# B&R Automation Studio project NAEUL004C00R13L518F00 (part 47)

### LF.typ - Do Not Change!!!
```iecst
(*2019-04-25*)
(**)
(*Action*)

TYPE
	eLFAction :
		(
		LFActIdle,
		LFActBGStartRun,
		LFActBGStopRun,
		LFActSyncPLCTm,
		LFActChgAllAuto,
		LFActChgAllMnl,
		LFActChgSeqAuto,
		LFActChgSeqMnl
		);
	eLFOPCUAStep :
		(
		LFOPCUAStepIncCntr,
		LFOPCUAStepChkHdls,
		LFOPCUAStepConnect,
		LFOPCUAStepWriteHdls,
		LFOPCUAStepReadHdls,
		LFOPCUAStepWrite,
		LFOPCUAStepRead,
		LFOPCUAStepStopChk
		);
	tyOPCUAHdlList : 	STRUCT
		a_dwHdls : ARRAY[0..MAX_INDEX_NODELIST]OF DWORD;
	END_STRUCT;
END_TYPE

(* *)

TYPE
	tyLFLeader1 : 	STRUCT
		In : tyLFLeaderIn1;
		Out : tyLFLeaderOut1;
	END_STRUCT;
	tyLFLeaderIn1 : 	STRUCT
		bPrep : BOOL;
		bEn : BOOL;
		bDis : BOOL;
	END_STRUCT;
	tyLFLeaderOut1 : 	STRUCT
		eStat : eLFAction;
		eStatus : eFBStatus;
		sStatTxt : STRING[100];
		a_tyFollowerInfo : ARRAY[1..c_diLFClntNum]OF tyLFFollowerInfo;
		a_tyFollowerToLeaderTag : ARRAY[1..c_diLFClntNum]OF tyLFFollowerToLeaderTag;
		tyAlmData : tyAlmDat;
	END_STRUCT;
END_TYPE

(* *)

TYPE
	tyLFFollower1 : 	STRUCT
		In : tyLFFollowerIn1;
		Out : tyLFFollowerOut1;
	END_STRUCT;
	tyLFFollowerIn1 : 	STRUCT
		bEn : BOOL;
		bDis : BOOL;
		bPrep : BOOL;
		bUSWidthChkSen : BOOL;
		bDSWidthChkSen : BOOL;
		sProgNm : STRING[15];
		sMagRcpNm : STRING[15];
	END_STRUCT;
	tyLFFollowerOut1 : 	STRUCT
		eStatus : eFBStatus;
		tyAlmData : tyAlmDat;
		tyInfoData : tyAlmDat;
		tyInfoData1 : tyAlmDat;
		bUSAllow : BOOL;
		bDSAllow : BOOL;
		bProdAccDataMnl : BOOL;
		bProdUpdtDataMnl : BOOL;
		bMagAccDataMnl : BOOL;
		eTimeAct : eTimeAction;
		dtTm : DATE_AND_TIME;
		bWaitRlsBrd : BOOL;
		tyUpdtProdRcp : tyProdRcpParam;
		bLdrSeqCtrlInActive : BOOL;
		tyLeaderInfo : tyLFLeaderInfo;
	END_STRUCT;
END_TYPE
```

### LF.var - Change By Project
```iecst
VAR
	p_LFLeader : UDINT;
	p_LFFollower : UDINT;
	p_Follower1 : UDINT;
	p_Follower2 : UDINT;
	g_sLFLeaderProgNm : STRING[15];
END_VAR
```

### Program Logical/LF/LFLeader (IEC, version 1.00.0) - 1.00.0 - NtHermes v5.00.0 , NtTCP v5.00.0 , NtMessage v5.00.0

#### Init.st - Change By Project
```iecst
(** 2019-04-30 **)
PROGRAM _INIT
	p_LFLeader := ADR(tylocalLFLeader.Out);

END_PROGRAM
```

#### Act_InputConfig.st - Change By Project
```iecst
ACTION Act_InputConfig:

	tylocalLFLeader.In.bPrep	:= g_tyNtParamCurr.bLFPrep;
	tylocalLFLeader.In.bDis 	:= g_tyStartUp.bRun OR (NOT g_tyNtParamCurr.bLFUsrSetPrep AND NOT g_tyNtParamCurr.bLeaderMc) OR (g_tyNtParamCurr.bLFUsrSetPrep AND NOT g_tyMcParamCurr.bLFLeaderMc);
	tylocalLFLeader.In.bEn		:= g_tyMcParamCurr.bLFLeaderMc;

	p_eAct ACCESS p_UILFLeaderAct;
	p_sReqProdRcpNm ACCESS p_ProdRcpCurrRcp0Nm;

	IF g_tyNtParamCurr.bLFProdWidth2Prep THEN
		p_diReqProdWidth ACCESS p_ProdRcpCurrRcp0Width2;
	ELSE
		p_diReqProdWidth ACCESS p_ProdRcpCurrRcp0Width;
	END_IF

	IF (g_tyUIOut.bUILeaderRun = TRUE) AND ((bRun1 = FALSE) OR (bRun2 = FALSE)) THEN
		bUILeaderStart	:= TRUE;
		bUILeaderStop	:= FALSE;
	END_IF

	IF (g_tyUIOut.bUILeaderRun = FALSE) AND ((bRun1 = TRUE) OR (bRun2 = TRUE)) THEN
		bUILeaderStart	:= FALSE;
		bUILeaderStop	:= TRUE;
	END_IF

	IF bUILeaderStart = TRUE THEN
		p_eAct	:= LFActBGStartRun;

		IF (tylocalLFLeader.Out.eStat = LFActBGStartRun) AND (tylocalLFLeader.Out.eStatus = Done) THEN
			p_eAct			:= LFActIdle;
			bUILeaderStart	:= FALSE;
		END_IF

	ELSIF bUILeaderStop = TRUE THEN
		p_eAct	:= LFActBGStopRun;

		IF (tylocalLFLeader.Out.eStat = LFActBGStopRun) AND (tylocalLFLeader.Out.eStatus = Done) THEN
			p_eAct			:= LFActIdle;
			bUILeaderStop	:= FALSE;
		END_IF

	END_IF
END_ACTION
```

#### Act_InitLocal.st - Do Not Change!!!
```iecst
(** 2020-08-06 **)
ACTION Act_InitLocal:

	//Input Reference Link To Local Variable
	p_eAct ACCESS ADR(eAct);

	p_sReqProdRcpNm ACCESS ADR(sReqProdRcpNm);
	p_diReqProdWidth ACCESS ADR(diReqProdWidth);
	p_sReqMagRcpNm ACCESS ADR(sReqMagRcpNm);

	p_sLeaderProgTagNm ACCESS ADR(sLeaderProgTagNm);
	p_sFollowerProgTagNm ACCESS ADR(sFollowerProgTagNm);

	p_bWidth2Prep ACCESS ADR(bWidth2Prep);
	p_bLFSeqStayActive ACCESS ADR(bLFSeqStayActive);

END_ACTION
```

#### Act_Initial.st - Do Not Change!!!
```iecst
ACTION Act_Initial:

	//Initial
	tylocalLFLeader.Out.sStatTxt	:= a_sStatText[tylocalLFLeader.Out.eStat];

	fbOnlineChk.pa_tyLeaderToFollowerTag	:= ADR(a_tyLeaderToFollowerTag);
	fbOnlineChk.pa_tyFollowerInfo	:= ADR(a_tyFollowerInfo);
	fbOnlineChk.tDlyTm				:= g_tyNtParamCurr.tLFLeaderOnlineChkDlyTm;
	fbOnlineChk(bEn := FALSE);

	fbSyncTm.pa_tyLeaderToFollowerTag	:= ADR(a_tyLeaderToFollowerTag);
	fbSyncTm.tDlyTm						:= g_tyNtParamCurr.tLFLeaderSetTmOffDlyTm;
	fbSyncTm(bEn := FALSE);

	fbChgAll.pa_tyLeaderToFollowerTag	:= ADR(a_tyLeaderToFollowerTag);
	fbChgAll(bEn := FALSE);

	fbChgSeq.pa_tyLeaderToFollowerTag	:= ADR(a_tyLeaderToFollowerTag);
	fbChgSeq(bEn := FALSE);

	fbBlkUSDS.pa_tyLeaderToFollowerTag	:= ADR(a_tyLeaderToFollowerTag);
	fbBlkUSDS(bEn := FALSE);

	fbDataUpdt.pa_tyLeaderToFollowerTag	:= ADR(a_tyLeaderToFollowerTag);
	fbDataUpdt(bEn := FALSE);

	fbConnect.tyOPCUAParam.sPort	:= '4840';
	fbConnect(bEn := FALSE);

	fbGetNodeHdlListWr.uiTagNmCnt			:= 17;
	fbGetNodeHdlListWr.a_sServerTagNm[0]	:= CONCAT(CONCAT('::' , p_sFollowerProgTagNm) , ':tyLeaderToFollowerTag.sReqProdRcpNm');
	fbGetNodeHdlListWr.a_sServerTagNm[1]	:= CONCAT(CONCAT('::' , p_sFollowerProgTagNm) , ':tyLeaderToFollowerTag.diReqProdRcpWidth');
	fbGetNodeHdlListWr.a_sServerTagNm[2]	:= CONCAT(CONCAT('::' , p_sFollowerProgTagNm) , ':tyLeaderToFollowerTag.sReqMagRcpNm');
	fbGetNodeHdlListWr.a_sServerTagNm[3]	:= CONCAT(CONCAT('::' , p_sFollowerProgTagNm) , ':tyLeaderToFollowerTag.bMnlAccData');
	fbGetNodeHdlListWr.a_sServerTagNm[4]	:= CONCAT(CONCAT('::' , p_sFollowerProgTagNm) , ':tyLeaderToFollowerTag.bBypassMnlAccData');
	fbGetNodeHdlListWr.a_sServerTagNm[5]	:= CONCAT(CONCAT('::' , p_sFollowerProgTagNm) , ':tyLeaderToFollowerTag.bBlkDS');
	fbGetNodeHdlListWr.a_sServerTagNm[6]	:= CONCAT(CONCAT('::' , p_sFollowerProgTagNm) , ':tyLeaderToFollowerTag.bBlkUS');
	fbGetNodeHdlListWr.a_sServerTagNm[7]	:= CONCAT(CONCAT('::' , p_sFollowerProgTagNm) , ':tyLeaderToFollowerTag.bSetTm');
	fbGetNodeHdlListWr.a_sServerTagNm[8]	:= CONCAT(CONCAT('::' , p_sFollowerProgTagNm) , ':tyLeaderToFollowerTag.dtTm');
	fbGetNodeHdlListWr.a_sServerTagNm[9]	:= CONCAT(CONCAT('::' , p_sFollowerProgTagNm) , ':tyLeaderToFollowerTag.uiTmZone');
	fbGetNodeHdlListWr.a_sServerTagNm[10]	:= CONCAT(CONCAT('::' , p_sFollowerProgTagNm) , ':tyLeaderToFollowerTag.bBypassWidthChk');
	fbGetNodeHdlListWr.a_sServerTagNm[11]	:= CONCAT(CONCAT('::' , p_sFollowerProgTagNm) , ':tyLeaderToFollowerTag.usiRunTm');
	fbGetNodeHdlListWr.a_sServerTagNm[12]	:= CONCAT(CONCAT('::' , p_sFollowerProgTagNm) , ':tyLeaderToFollowerTag.bProdNameUSWarn');
	fbGetNodeHdlListWr.a_sServerTagNm[13]	:= CONCAT(CONCAT('::' , p_sFollowerProgTagNm) , ':tyLeaderToFollowerTag.bProdNameDSWarn');
	fbGetNodeHdlListWr.a_sServerTagNm[14]	:= CONCAT(CONCAT('::' , p_sFollowerProgTagNm) , ':tyLeaderToFollowerTag.bProdWidthUSWarn');
	fbGetNodeHdlListWr.a_sServerTagNm[15]	:= CONCAT(CONCAT('::' , p_sFollowerProgTagNm) , ':tyLeaderToFollowerTag.bProdWidthDSWarn');
	fbGetNodeHdlListWr.a_sServerTagNm[16]	:= CONCAT(CONCAT('::' , p_sFollowerProgTagNm) , ':tyLeaderToFollowerTag.bLeaderSeqCtrlInActive');
	fbGetNodeHdlListWr(bEn := FALSE);

	fbGetNodeHdlListRd.uiTagNmCnt			:= 14;
	fbGetNodeHdlListRd.a_sServerTagNm[0]	:= CONCAT(CONCAT('::' , p_sFollowerProgTagNm) , ':tyFollowerToLeaderTag.sCurrProdRcp');
	fbGetNodeHdlListRd.a_sServerTagNm[1]	:= CONCAT(CONCAT('::' , p_sFollowerProgTagNm) , ':tyFollowerToLeaderTag.diCurrProdWidthUS');
	fbGetNodeHdlListRd.a_sServerTagNm[2]	:= CONCAT(CONCAT('::' , p_sFollowerProgTagNm) , ':tyFollowerToLeaderTag.sCurrMagRcp');
	fbGetNodeHdlListRd.a_sServerTagNm[3]	:= CONCAT(CONCAT('::' , p_sFollowerProgTagNm) , ':tyFollowerToLeaderTag.sIPAddr');
	fbGetNodeHdlListRd.a_sServerTagNm[4]	:= CONCAT(CONCAT('::' , p_sFollowerProgTagNm) , ':tyFollowerToLeaderTag.sMcNm');
	fbGetNodeHdlListRd.a_sServerTagNm[5]	:= CONCAT(CONCAT('::' , p_sFollowerProgTagNm) , ':tyFollowerToLeaderTag.bSectionLeader');
	fbGetNodeHdlListRd.a_sServerTagNm[6]	:= CONCAT(CONCAT('::' , p_sFollowerProgTagNm) , ':tyFollowerToLeaderTag.usiRunTm');
	fbGetNodeHdlListRd.a_sServerTagNm[7]	:= CONCAT(CONCAT('::' , p_sFollowerProgTagNm) , ':tyFollowerToLeaderTag.bProdRcpErr');
	fbGetNodeHdlListRd.a_sServerTagNm[8]	:= CONCAT(CONCAT('::' , p_sFollowerProgTagNm) , ':tyFollowerToLeaderTag.bProdWidthErr');
	fbGetNodeHdlListRd.a_sServerTagNm[9]	:= CONCAT(CONCAT('::' , p_sFollowerProgTagNm) , ':tyFollowerToLeaderTag.bMagRcpErr');
	fbGetNodeHdlListRd.a_sServerTagNm[10]	:= CONCAT(CONCAT('::' , p_sFollowerProgTagNm) , ':tyFollowerToLeaderTag.bSyncTmErr');
	fbGetNodeHdlListRd.a_sServerTagNm[11]	:= CONCAT(CONCAT('::' , p_sFollowerProgTagNm) , ':tyFollowerToLeaderTag.diCurrProdWidthDS');
	fbGetNodeHdlListRd.a_sServerTagNm[12]	:= CONCAT(CONCAT('::' , p_sFollowerProgTagNm) , ':tyFollowerToLeaderTag.eCurrMachineStat');
	fbGetNodeHdlListRd.a_sServerTagNm[13]	:= CONCAT(CONCAT('::' , p_sFollowerProgTagNm) , ':tyFollowerToLeaderTag.bProdChgOverActive');
	fbGetNodeHdlListRd(bEn := FALSE);

	fbWriteList.uiTagNmCnt	:= 17;
	fbWriteList(bEn := FALSE);

	fbReadList.uiTagNmCnt	:= 14;
	fbReadList(bEn := FALSE);

	fbDisconnect(bEn := FALSE);

END_ACTION
```

#### Act_Main.st - Do Not Change!!!
```iecst
ACTION Act_Main:

		//Set p_eAct
	IF tylocalLFLeader.Out.eStatus = Idle OR tylocalLFLeader.Out.eStatus = Busy OR tylocalLFLeader.Out.eStatus = Done THEN
		tylocalLFLeader.Out.eStat	:= p_eAct;
	END_IF

	IF eStatOld <> tylocalLFLeader.Out.eStat THEN
		fbSyncTm(bEn := FALSE);
		fbChgAll(bEn := FALSE);
		fbChgSeq(bEn := FALSE);

		tylocalLFLeader.Out.sStatTxt	:= a_sStatText[tylocalLFLeader.Out.eStat];

		eStatOld	:= tylocalLFLeader.Out.eStat;

		tylocalLFLeader.Out.eStatus		:= Busy;
	END_IF

	//Main
	CASE tylocalLFLeader.Out.eStat OF

		LFActIdle:
			tylocalLFLeader.Out.eStatus	:= Idle;

		LFActBGStartRun:
			IF tylocalLFLeader.Out.eStatus = Idle OR tylocalLFLeader.Out.eStatus = Busy THEN

				bRun1		:= TRUE;
				bRun2		:= TRUE;
				bStop		:= FALSE;
				bStop1Done	:= FALSE;
				bStop2Done	:= FALSE;
				tylocalLFLeader.Out.eStatus		:= Done;

			END_IF

		LFActBGStopRun:
			IF tylocalLFLeader.Out.eStatus = Idle OR tylocalLFLeader.Out.eStatus = Busy THEN

				tylocalLFLeader.Out.eStatus	:= Busy;

				bStop	:= TRUE;

				IF bStop1Done AND bStop2Done THEN

					bRun1		:= FALSE;
					bRun2		:= FALSE;
					bStop		:= FALSE;
					bStop1Done	:= FALSE;
					bStop2Done	:= FALSE;
					tylocalLFLeader.Out.eStatus		:= Done;

				END_IF

			END_IF

		LFActSyncPLCTm:
			IF tylocalLFLeader.Out.eStatus = Idle OR tylocalLFLeader.Out.eStatus = Busy THEN

				IF bRun1 AND bRun2 THEN
					tylocalLFLeader.Out.eStatus	:= Busy;

					fbSyncTm.dtCurrDT		:= g_tyTime.dtCurrDT;
					fbSyncTm.diMcNum		:= diMcNum;
					fbSyncTm(bEn := TRUE);

					IF fbSyncTm.udiStatus = 0 THEN
						tylocalLFLeader.Out.eStatus	:= Done;
					ELSIF fbSyncTm.udiStatus < 65534 THEN
						tylocalLFLeader.Out.eStatus		:= Error;
						udiStatus	:= fbSyncTm.udiStatus;
					END_IF

				ELSE
					tylocalLFLeader.Out.eStatus		:= Error;
					udiStatus	:= 10000;	//Background Not Running While Calling Sync PLC Tm
				END_IF

			END_IF

		LFActChgAllAuto:
			IF tylocalLFLeader.Out.eStatus = Idle OR tylocalLFLeader.Out.eStatus = Busy THEN

				IF bRun1 AND bRun2 THEN
					tylocalLFLeader.Out.eStatus	:= Busy;

					fbChgAll.bChgAuto					:= TRUE;
					fbChgAll.a_bOnline					:= g_tyMcParamCurr.a_bLFOnline;;
					fbChgAll.a_tyFollowerToLeaderTag	:= a_tyFollowerToLeaderTag;
					fbChgAll.sReqProdRcpNm				:= p_sReqProdRcpNm;
					fbChgAll.diReqProdRcpWidth			:= p_diReqProdWidth;
					fbChgAll.sReqMagRcpNm				:= p_sReqMagRcpNm;
					fbChgAll.diMcNum					:= diMcNum;
					fbChgAll(bEn := TRUE);

					IF fbChgAll.udiStatus = 0 THEN
						tylocalLFLeader.Out.eStatus	:= Done;
					ELSIF fbChgAll.udiStatus < 65534 THEN
						tylocalLFLeader.Out.eStatus		:= Error;
						udiStatus	:= fbChgAll.udiStatus;
					END_IF

				ELSE
					tylocalLFLeader.Out.eStatus		:= Error;
					udiStatus	:= 10001;	//Background Not Running While Changing All Recipe Automatically
				END_IF

			END_IF

		LFActChgAllMnl:
			IF tylocalLFLeader.Out.eStatus = Idle OR tylocalLFLeader.Out.eStatus = Busy THEN

				IF bRun1 AND bRun2 THEN
					tylocalLFLeader.Out.eStatus	:= Busy;

					fbChgAll.bChgAuto					:= FALSE;
					fbChgAll.a_bOnline					:= g_tyMcParamCurr.a_bLFOnline;
					fbChgAll.a_tyFollowerToLeaderTag	:= a_tyFollowerToLeaderTag;
					fbChgAll.sReqProdRcpNm				:= p_sReqProdRcpNm;
					fbChgAll.diReqProdRcpWidth			:= p_diReqProdWidth;
					fbChgAll.sReqMagRcpNm				:= p_sReqMagRcpNm;
					fbChgAll.diMcNum					:= diMcNum;
					fbChgAll(bEn := TRUE);

					IF fbChgAll.udiStatus = 0 THEN
						tylocalLFLeader.Out.eStatus	:= Done;
					ELSIF fbChgAll.udiStatus < 65534 THEN
						tylocalLFLeader.Out.eStatus		:= Error;
						udiStatus	:= fbChgAll.udiStatus;
					END_IF

				ELSE
					tylocalLFLeader.Out.eStatus		:= Error;
					udiStatus	:= 10002;	//Background Not Running While Changing All Recipe Manually
				END_IF

			END_IF

		LFActChgSeqAuto:
			IF tylocalLFLeader.Out.eStatus = Idle OR tylocalLFLeader.Out.eStatus = Busy THEN

				IF bRun1 AND bRun2 THEN
					tylocalLFLeader.Out.eStatus	:= Busy;

					fbChgSeq.bChgAuto					:= TRUE;
					fbChgSeq.a_bOnline					:= g_tyMcParamCurr.a_bLFOnline;;
					fbChgSeq.a_tyFollowerToLeaderTag	:= a_tyFollowerToLeaderTag;
					fbChgSeq.sReqProdRcpNm				:= p_sReqProdRcpNm;
					fbChgSeq.diReqProdRcpWidth			:= p_diReqProdWidth;
					fbChgSeq.sReqMagRcpNm				:= p_sReqMagRcpNm;
					fbChgSeq.diMcNum					:= diMcNum;
					fbChgSeq(bEn := TRUE);

					IF fbChgSeq.udiStatus = 0 THEN
						tylocalLFLeader.Out.eStatus	:= Done;
					ELSIF fbChgSeq.udiStatus < 65534 THEN
						tylocalLFLeader.Out.eStatus		:= Error;
						udiStatus	:= fbChgSeq.udiStatus;
					END_IF

				ELSE
					tylocalLFLeader.Out.eStatus		:= Error;
					udiStatus	:= 10003;	//Background Not Running While Changing Recipe In Sequence Automatically
				END_IF

			END_IF

		LFActChgSeqMnl:
			IF tylocalLFLeader.Out.eStatus = Idle OR tylocalLFLeader.Out.eStatus = Busy THEN

				IF bRun1 AND bRun2 THEN
					tylocalLFLeader.Out.eStatus	:= Busy;

					fbChgSeq.bChgAuto					:= FALSE;
					fbChgSeq.a_bOnline					:= g_tyMcParamCurr.a_bLFOnline;;
					fbChgSeq.a_tyFollowerToLeaderTag	:= a_tyFollowerToLeaderTag;
					fbChgSeq.sReqProdRcpNm				:= p_sReqProdRcpNm;
					fbChgSeq.diReqProdRcpWidth			:= p_diReqProdWidth;
					fbChgSeq.sReqMagRcpNm				:= p_sReqMagRcpNm;
					fbChgSeq.diMcNum					:= diMcNum;
					fbChgSeq(bEn := TRUE);

					IF fbChgSeq.udiStatus = 0 THEN
						tylocalLFLeader.Out.eStatus	:= Done;
					ELSIF fbChgSeq.udiStatus < 65534 THEN
						tylocalLFLeader.Out.eStatus		:= Error;
						udiStatus	:= fbChgSeq.udiStatus;
					END_IF

				ELSE
					tylocalLFLeader.Out.eStatus		:= Error;
					udiStatus	:= 10004;	//Background Not Running While Changing Recipe In Sequence Manually
				END_IF

			END_IF

	END_CASE

END_ACTION
```

#### Act_Background.st - Do Not Change!!!
```iecst
ACTION Act_Background:

	IF EDGEPOS(bRun1 AND bRun2) THEN

		FOR di := 1 TO c_diLFClntNum DO
			IF g_tyMcParamCurr.a_sLFIPAddr[di] = '' THEN
				diMcNum	:= di - 1;
				EXIT;
			END_IF
		END_FOR

	END_IF

	Act_Background_OPCUA;
	Act_Background_Process;
	Act_Background_Disconnect;

END_ACTION
```

#### Act_Background_OPCUA.st - Do Not Change!!!
```iecst
ACTION Act_Background_OPCUA:

	IF bRun1 = TRUE THEN

		CASE eOPCUAStep OF

			LFOPCUAStepIncCntr:
				udiNodeCntr	:= udiNodeCntr + 1;

				IF udiNodeCntr > c_diLFClntNum THEN
					udiNodeCntr	:= 1;
				END_IF

				eOPCUAStep	:= LFOPCUAStepChkHdls;

			LFOPCUAStepChkHdls:
				IF g_tyMcParamCurr.a_sLFIPAddr[udiNodeCntr] <> '' THEN
					IF g_tyMcParamCurr.a_bLFOnline[udiNodeCntr] = TRUE THEN
						IF a_dwConnectionHdl[udiNodeCntr] <> 0 THEN
							IF a_bNodeWr[udiNodeCntr] = TRUE THEN
								IF a_bNodeRd[udiNodeCntr] = TRUE THEN
									eOPCUAStep	:= LFOPCUAStepWrite;
								ELSE
									eOPCUAStep	:= LFOPCUAStepReadHdls;
								END_IF
							ELSE
								eOPCUAStep	:= LFOPCUAStepWriteHdls;
							END_IF
						ELSE
							eOPCUAStep	:= LFOPCUAStepConnect;
						END_IF
					ELSE
						eOPCUAStep	:= LFOPCUAStepIncCntr;
					END_IF
				ELSE
					udiNodeCntr	:= 0;
					eOPCUAStep	:= LFOPCUAStepStopChk;
				END_IF

			LFOPCUAStepConnect:
				fbConnect.tyOPCUAParam.sIPAddr	:= g_tyMcParamCurr.a_sLFIPAddr[udiNodeCntr];
				fbConnect(bEn := TRUE);

				IF fbConnect.udiStatus = 0 THEN
					a_dwConnectionHdl[udiNodeCntr]	:= fbConnect.dwConnectionHdl;
					fbConnect(bEn := FALSE);
					eOPCUAStep	:= LFOPCUAStepWriteHdls;
				ELSIF fbConnect.udiStatus < 65534 THEN
					a_dwConnectionHdl[udiNodeCntr]	:= 0;
					fbConnect(bEn := FALSE);
					eOPCUAStep	:= LFOPCUAStepStopChk;
				END_IF

			LFOPCUAStepWriteHdls:
				fbGetNodeHdlListWr.dwConnectionHdl	:= a_dwConnectionHdl[udiNodeCntr];
				fbGetNodeHdlListWr(bEn := TRUE);

				IF fbGetNodeHdlListWr.udiStatus = 0 THEN
					a_bNodeWr[udiNodeCntr]				:= TRUE;
					a_tyWriteHdls[udiNodeCntr].a_dwHdls	:= fbGetNodeHdlListWr.a_dwNodeHdlList;
					fbGetNodeHdlListWr(bEn := FALSE);
					eOPCUAStep	:= LFOPCUAStepReadHdls;
				ELSIF fbGetNodeHdlListWr.udiStatus < 65534 THEN
					a_bNodeWr[udiNodeCntr]	:= FALSE;
					fbGetNodeHdlListWr(bEn := FALSE);
					eOPCUAStep	:= LFOPCUAStepStopChk;
				END_IF

			LFOPCUAStepReadHdls:
				fbGetNodeHdlListRd.dwConnectionHdl	:= a_dwConnectionHdl[udiNodeCntr];
				fbGetNodeHdlListRd(bEn := TRUE);

				IF fbGetNodeHdlListRd.udiStatus = 0 THEN
					a_bNodeRd[udiNodeCntr]				:= TRUE;
					a_tyReadHdls[udiNodeCntr].a_dwHdls	:= fbGetNodeHdlListRd.a_dwNodeHdlList;
					fbGetNodeHdlListRd(bEn := FALSE);
					eOPCUAStep	:= LFOPCUAStepWrite;
				ELSIF fbGetNodeHdlListRd.udiStatus < 65534 THEN
					a_bNodeRd[udiNodeCntr]	:= FALSE;
					fbGetNodeHdlListRd(bEn := FALSE);
					eOPCUAStep	:= LFOPCUAStepStopChk;
				END_IF

			LFOPCUAStepWrite:
				fbWriteList.dwConnectionHdl		:= a_dwConnectionHdl[udiNodeCntr];
				fbWriteList.a_dwNodeHdlList		:= a_tyWriteHdls[udiNodeCntr].a_dwHdls;
				sNodeCntr						:= UDINT_TO_STRING(udiNodeCntr);
				fbWriteList.a_sClientTagNm[0]	:= CONCAT(CONCAT(CONCAT(CONCAT('::' , p_sLeaderProgTagNm) , ':a_tyLeaderToFollowerTag[') , sNodeCntr) , '].sReqProdRcpNm');
				fbWriteList.a_sClientTagNm[1]	:= CONCAT(CONCAT(CONCAT(CONCAT('::' , p_sLeaderProgTagNm) , ':a_tyLeaderToFollowerTag[') , sNodeCntr) , '].diReqProdRcpWidth');
				fbWriteList.a_sClientTagNm[2]	:= CONCAT(CONCAT(CONCAT(CONCAT('::' , p_sLeaderProgTagNm) , ':a_tyLeaderToFollowerTag[') , sNodeCntr) , '].sReqMagRcpNm');
				fbWriteList.a_sClientTagNm[3]	:= CONCAT(CONCAT(CONCAT(CONCAT('::' , p_sLeaderProgTagNm) , ':a_tyLeaderToFollowerTag[') , sNodeCntr) , '].bMnlAccData');
				fbWriteList.a_sClientTagNm[4]	:= CONCAT(CONCAT(CONCAT(CONCAT('::' , p_sLeaderProgTagNm) , ':a_tyLeaderToFollowerTag[') , sNodeCntr) , '].bBypassMnlAccData');
				fbWriteList.a_sClientTagNm[5]	:= CONCAT(CONCAT(CONCAT(CONCAT('::' , p_sLeaderProgTagNm) , ':a_tyLeaderToFollowerTag[') , sNodeCntr) , '].bBlkDS');
				fbWriteList.a_sClientTagNm[6]	:= CONCAT(CONCAT(CONCAT(CONCAT('::' , p_sLeaderProgTagNm) , ':a_tyLeaderToFollowerTag[') , sNodeCntr) , '].bBlkUS');
				fbWriteList.a_sClientTagNm[7]	:= CONCAT(CONCAT(CONCAT(CONCAT('::' , p_sLeaderProgTagNm) , ':a_tyLeaderToFollowerTag[') , sNodeCntr) , '].bSetTm');
				fbWriteList.a_sClientTagNm[8]	:= CONCAT(CONCAT(CONCAT(CONCAT('::' , p_sLeaderProgTagNm) , ':a_tyLeaderToFollowerTag[') , sNodeCntr) , '].dtTm');
				fbWriteList.a_sClientTagNm[9]	:= CONCAT(CONCAT(CONCAT(CONCAT('::' , p_sLeaderProgTagNm) , ':a_tyLeaderToFollowerTag[') , sNodeCntr) , '].uiTmZone');
				fbWriteList.a_sClientTagNm[10]	:= CONCAT(CONCAT(CONCAT(CONCAT('::' , p_sLeaderProgTagNm) , ':a_tyLeaderToFollowerTag[') , sNodeCntr) , '].bBypassWidthChk');
				fbWriteList.a_sClientTagNm[11]	:= CONCAT(CONCAT(CONCAT(CONCAT('::' , p_sLeaderProgTagNm) , ':a_tyLeaderToFollowerTag[') , sNodeCntr) , '].usiRunTm');
				fbWriteList.a_sClientTagNm[12]	:= CONCAT(CONCAT(CONCAT(CONCAT('::' , p_sLeaderProgTagNm) , ':a_tyLeaderToFollowerTag[') , sNodeCntr) , '].bProdNameUSWarn');
				fbWriteList.a_sClientTagNm[13]	:= CONCAT(CONCAT(CONCAT(CONCAT('::' , p_sLeaderProgTagNm) , ':a_tyLeaderToFollowerTag[') , sNodeCntr) , '].bProdNameDSWarn');
				fbWriteList.a_sClientTagNm[14]	:= CONCAT(CONCAT(CONCAT(CONCAT('::' , p_sLeaderProgTagNm) , ':a_tyLeaderToFollowerTag[') , sNodeCntr) , '].bProdWidthUSWarn');
				fbWriteList.a_sClientTagNm[15]	:= CONCAT(CONCAT(CONCAT(CONCAT('::' , p_sLeaderProgTagNm) , ':a_tyLeaderToFollowerTag[') , sNodeCntr) , '].bProdWidthDSWarn');
				fbWriteList.a_sClientTagNm[16]	:= CONCAT(CONCAT(CONCAT(CONCAT('::' , p_sLeaderProgTagNm) , ':a_tyLeaderToFollowerTag[') , sNodeCntr) , '].bLeaderSeqCtrlInActive');
				fbWriteList(bEn := TRUE);

				IF fbWriteList.udiStatus = 0 THEN
					fbWriteList(bEn := FALSE);
					eOPCUAStep	:= LFOPCUAStepRead;
				ELSIF fbWriteList.udiStatus < 65534 THEN
					fbWriteList(bEn := FALSE);
					eOPCUAStep	:= LFOPCUAStepStopChk;
				END_IF

			LFOPCUAStepRead:
				fbReadList.dwConnectionHdl		:= a_dwConnectionHdl[udiNodeCntr];
				fbReadList.a_dwNodeHdlList		:= a_tyReadHdls[udiNodeCntr].a_dwHdls;
				sNodeCntr						:= UDINT_TO_STRING(udiNodeCntr);
				fbReadList.a_sClientTagNm[0]	:= CONCAT(CONCAT(CONCAT(CONCAT('::' , p_sLeaderProgTagNm) , ':a_tyFollowerToLeaderTag[') , sNodeCntr) , '].sCurrProdRcp');
				fbReadList.a_sClientTagNm[1]	:= CONCAT(CONCAT(CONCAT(CONCAT('::' , p_sLeaderProgTagNm) , ':a_tyFollowerToLeaderTag[') , sNodeCntr) , '].diCurrProdWidthUS');
				fbReadList.a_sClientTagNm[2]	:= CONCAT(CONCAT(CONCAT(CONCAT('::' , p_sLeaderProgTagNm) , ':a_tyFollowerToLeaderTag[') , sNodeCntr) , '].sCurrMagRcp');
				fbReadList.a_sClientTagNm[3]	:= CONCAT(CONCAT(CONCAT(CONCAT('::' , p_sLeaderProgTagNm) , ':a_tyFollowerToLeaderTag[') , sNodeCntr) , '].sIPAddr');
				fbReadList.a_sClientTagNm[4]	:= CONCAT(CONCAT(CONCAT(CONCAT('::' , p_sLeaderProgTagNm) , ':a_tyFollowerToLeaderTag[') , sNodeCntr) , '].sMcNm');
				fbReadList.a_sClientTagNm[5]	:= CONCAT(CONCAT(CONCAT(CONCAT('::' , p_sLeaderProgTagNm) , ':a_tyFollowerToLeaderTag[') , sNodeCntr) , '].bSectionLeader');
				fbReadList.a_sClientTagNm[6]	:= CONCAT(CONCAT(CONCAT(CONCAT('::' , p_sLeaderProgTagNm) , ':a_tyFollowerToLeaderTag[') , sNodeCntr) , '].usiRunTm');
				fbReadList.a_sClientTagNm[7]	:= CONCAT(CONCAT(CONCAT(CONCAT('::' , p_sLeaderProgTagNm) , ':a_tyFollowerToLeaderTag[') , sNodeCntr) , '].bProdRcpErr');
				fbReadList.a_sClientTagNm[8]	:= CONCAT(CONCAT(CONCAT(CONCAT('::' , p_sLeaderProgTagNm) , ':a_tyFollowerToLeaderTag[') , sNodeCntr) , '].bProdWidthErr');
				fbReadList.a_sClientTagNm[9]	:= CONCAT(CONCAT(CONCAT(CONCAT('::' , p_sLeaderProgTagNm) , ':a_tyFollowerToLeaderTag[') , sNodeCntr) , '].bMagRcpErr');
				fbReadList.a_sClientTagNm[10]	:= CONCAT(CONCAT(CONCAT(CONCAT('::' , p_sLeaderProgTagNm) , ':a_tyFollowerToLeaderTag[') , sNodeCntr) , '].bSyncTmErr');
				fbReadList.a_sClientTagNm[11]	:= CONCAT(CONCAT(CONCAT(CONCAT('::' , p_sLeaderProgTagNm) , ':a_tyFollowerToLeaderTag[') , sNodeCntr) , '].diCurrProdWidthDS');
				fbReadList.a_sClientTagNm[12]	:= CONCAT(CONCAT(CONCAT(CONCAT('::' , p_sLeaderProgTagNm) , ':a_tyFollowerToLeaderTag[') , sNodeCntr) , '].eCurrMachineStat');
				fbReadList.a_sClientTagNm[13]	:= CONCAT(CONCAT(CONCAT(CONCAT('::' , p_sLeaderProgTagNm) , ':a_tyFollowerToLeaderTag[') , sNodeCntr) , '].bProdChgOverActive');
				fbReadList(bEn := TRUE);

				IF fbReadList.udiStatus = 0 THEN
					fbReadList(bEn := FALSE);
					eOPCUAStep	:= LFOPCUAStepStopChk;
				ELSIF fbReadList.udiStatus < 65534 THEN
					fbReadList(bEn := FALSE);
					eOPCUAStep	:= LFOPCUAStepStopChk;
				END_IF

			LFOPCUAStepStopChk:
				IF bStop AND bStop2Done THEN
					IF bCntr = FALSE THEN
						bCntr	:= TRUE;
					ELSE
						bStop1Done	:= TRUE;
						bCntr		:= FALSE;
					END_IF
				ELSE
					bCntr	:= FALSE;
				END_IF

				eOPCUAStep	:= LFOPCUAStepIncCntr;

		END_CASE

	END_IF

END_ACTION
```

#### Act_Background_Process.st - Do Not Change!!!
```iecst
ACTION Act_Background_Process:

	IF bRun2 = TRUE AND bStop = FALSE THEN
		fbOnlineChk.a_bOnline				:= g_tyMcParamCurr.a_bLFOnline;
		fbOnlineChk.a_tyFollowerToLeaderTag	:= a_tyFollowerToLeaderTag;
		fbOnlineChk.diMcNum					:= diMcNum;
		fbOnlineChk(bEn := TRUE);

		fbBlkUSDS.a_tyFollowerToLeaderTag	:= a_tyFollowerToLeaderTag;
		fbBlkUSDS.diBeforeOven1			:= g_tyMcParamCurr.diLFMcIdxBeforeOven;
		fbBlkUSDS.diAfterOven1			:= g_tyMcParamCurr.diLFMcIdxAfterOven;
		fbBlkUSDS.diBeforeOven2			:= g_tyMcParamCurr.diLFMcIdxBeforeOven2;
		fbBlkUSDS.diAfterOven2			:= g_tyMcParamCurr.diLFMcIdxAfterOven2;
		fbBlkUSDS.diMcNum				:= diMcNum;
		fbBlkUSDS.pa_bLFOnline			:= g_tyMcParamCurr.a_bLFOnline;
		fbBlkUSDS.bSeqMode				:= (tylocalLFLeader.Out.eStat= LFActChgSeqAuto) OR (tylocalLFLeader.Out.eStat= LFActChgSeqMnl);
		fbBlkUSDS(bEn := TRUE);

		fbDataUpdt.a_bOnline			:= g_tyMcParamCurr.a_bLFOnline;
		fbDataUpdt.diMcNum				:= diMcNum;
		fbDataUpdt(bEn := TRUE);

	ELSIF bStop = TRUE THEN
		fbOnlineChk(bEn := FALSE);
		fbBlkUSDS(bEn := FALSE);
		fbDataUpdt(bEn := FALSE);
		bStop2Done	:= TRUE;

	END_IF

END_ACTION
```

#### Act_Background_Disconnect.st - Do Not Change!!!
```iecst
ACTION Act_Background_Disconnect:

	IF (memcmp(ADR(g_tyMcParamCurr.a_sLFIPAddr) , ADR(a_sLFIPAddrOld) , SIZEOF(a_sLFIPAddrOld)) <> 0) AND (bDisconnecting = FALSE) THEN
		FOR di := 1 TO c_diLFClntNum DO

			IF g_tyMcParamCurr.a_sLFIPAddr[di] <> a_sLFIPAddrOld[di] THEN
				diDisconnectIdx	:= di;
				bDisconnecting	:= TRUE;
				EXIT;
			END_IF

		END_FOR
	END_IF

	IF bDisconnecting = TRUE THEN

		IF a_dwConnectionHdl[diDisconnectIdx] <> 0 THEN
			fbDisconnect.dwConnectionHdl	:= a_dwConnectionHdl[diDisconnectIdx];
			fbDisconnect(bEn := TRUE);

			IF fbDisconnect.udiStatus = 0 THEN
				a_dwConnectionHdl[diDisconnectIdx]	:= 0;
				a_bNodeWr[diDisconnectIdx]			:= FALSE;
				a_bNodeRd[diDisconnectIdx]			:= FALSE;
				memset(ADR(a_tyFollowerToLeaderTag[diDisconnectIdx]) , 0 , SIZEOF(a_tyFollowerToLeaderTag[diDisconnectIdx]));
				fbDisconnect(bEn := FALSE);

				a_sLFIPAddrOld[diDisconnectIdx]	:= g_tyMcParamCurr.a_sLFIPAddr[diDisconnectIdx];
				bDisconnecting						:= FALSE;

			ELSIF fbDisconnect.udiStatus < 65534 THEN
				a_dwConnectionHdl[diDisconnectIdx]	:= 0;
				a_bNodeWr[diDisconnectIdx]			:= FALSE;
				a_bNodeRd[diDisconnectIdx]			:= FALSE;
				memset(ADR(a_tyFollowerToLeaderTag[diDisconnectIdx]) , 0 , SIZEOF(a_tyFollowerToLeaderTag[diDisconnectIdx]));
				fbDisconnect(bEn := FALSE);

				a_sLFIPAddrOld[diDisconnectIdx]	:= g_tyMcParamCurr.a_sLFIPAddr[diDisconnectIdx];
				bDisconnecting						:= FALSE;

			END_IF

		ELSE
			a_bNodeWr[diDisconnectIdx]	:= FALSE;
			a_bNodeRd[diDisconnectIdx]	:= FALSE;
			memset(ADR(a_tyFollowerToLeaderTag[diDisconnectIdx]) , 0 , SIZEOF(a_tyFollowerToLeaderTag[diDisconnectIdx]));

			a_sLFIPAddrOld[diDisconnectIdx]	:= g_tyMcParamCurr.a_sLFIPAddr[diDisconnectIdx];
			bDisconnecting						:= FALSE;

		END_IF

	END_IF

END_ACTION
```

#### Act_Alarm.st - Do Not Change!!!
```iecst
ACTION Act_Alarm:

	IF g_tyRstErrOut.udiRstErr <> udiRstErrOld THEN
		bRstErr			:= TRUE;
		udiRstErrOld	:= g_tyRstErrOut.udiRstErr;
	ELSE
		bRstErr			:= FALSE;
	END_IF

	//Reset Error
	IF (tylocalLFLeader.Out.eStatus = Error) AND bRstErr THEN
		p_eAct	:= LFActIdle;
		tylocalLFLeader.Out.eStat	:= LFActIdle;
	END_IF

	//Error
	IF EDGEPOS(tylocalLFLeader.Out.eStatus = Error) THEN

		tylocalLFLeader.Out.tyAlmData.udiCode		:= udiStatus;
		tylocalLFLeader.Out.tyAlmData.eSeverity		:= AlmSeverityError;
		tylocalLFLeader.Out.tyAlmData.udiRunTime	:= tyAlmData.udiRunTime + 1;
		tylocalLFLeader.Out.tyAlmData.bAlm			:= TRUE;
		tylocalLFLeader.Out.tyAlmData.udiModuleNum  := udiModuleNum;
		g_sLFLeaderProgNm		:= g_tyNtParamCurr.sLFLeaderProgNm;

	ELSIF bRstErr AND (tyAlmData.udiCode <> 0) THEN

		tylocalLFLeader.Out.tyAlmData.udiCode	:= 0;
		tylocalLFLeader.Out.tyAlmData.eSeverity	:= AlmSeverityNA;
		tylocalLFLeader.Out.tyAlmData.bAlm		:= FALSE;
		tylocalLFLeader.Out.sStatTxt	:= a_sStatText[tylocalLFLeader.Out.eStat];

	END_IF

END_ACTION
```

#### Local.var - Do Not Change!!!
```iecst
(*Reference Data Points*)
VAR
	p_eAct : REFERENCE TO eLFAction;
	p_sReqProdRcpNm : REFERENCE TO STRING[254];
	p_diReqProdWidth : REFERENCE TO DINT;
	p_sReqMagRcpNm : REFERENCE TO STRING[15];
	p_sLeaderProgTagNm : REFERENCE TO STRING[15];
	p_sFollowerProgTagNm : REFERENCE TO STRING[15];
END_VAR
(**)
VAR
	tylocalLFLeader : tyLFLeader1;
	a_sStatText : ARRAY[0..50] OF STRING[200] := ['Idling','Background Starting Operations','Background Stopping Operations','Synchronizing PLC Time','Changing All Recipe Automatically','Changing All Recipe Manually','Changing Recipe In Sequence Automatically','Changing Recipe In Sequence Manually',43('')];
END_VAR
(**)
(*Local Alarm*)
VAR
	tyAlmData : tyAlmDat;
END_VAR
(**)
(*Local Output*)
VAR
	a_tyFollowerInfo : ARRAY[1..c_diLFClntNum] OF tyLFFollowerInfo;
	a_tyFollowerToLeaderTag : ARRAY[1..c_diLFClntNum] OF tyLFFollowerToLeaderTag;
END_VAR
(**)
(*Local Input*)
VAR
	eAct : eLFAction;
	udiStatus : UDINT;
	sReqProdRcpNm : STRING[254];
	diReqProdWidth : DINT;
	sReqMagRcpNm : STRING[15];
	sLeaderProgTagNm : STRING[15] := 'LFLeader';
	sFollowerProgTagNm : STRING[15] := 'LFFollower';
	bUILeaderStart : BOOL;
	bUILeaderStop : BOOL;
END_VAR
(**)
VAR
	bRstErr : BOOL;
	udiRstErrOld : UDINT;
	bInitDone : BOOL;
	bInitialDone : BOOL;
	bRun1 : BOOL;
	bRun2 : BOOL;
	bStop : BOOL;
	bStop1Done : BOOL;
	bStop2Done : BOOL;
	bCntr : BOOL;
	di : DINT;
	diDisconnectIdx : DINT := 1;
	diMcNum : DINT;
	a_sLFIPAddrOld : ARRAY[1..c_diLFClntNum] OF STRING[15];
	bDisconnecting : BOOL;
	eStatOld : eLFAction := LFActIdle;
	a_tyLeaderToFollowerTag : ARRAY[1..c_diLFClntNum] OF tyLFLeaderToFollowerTag;
	fbOnlineChk : fbLFLeaderOnlineChk;
	fbSyncTm : fbLFLeaderSyncTm;
	fbChgAll : fbLFLeaderChgAll;
	fbChgSeq : fbLFLeaderChgSeq;
	fbBlkUSDS : fbLFLeaderBlkUSDS;
	fbDataUpdt : fbLFLeaderDataUpdt;
	udiNodeCntr : UDINT;
	sNodeCntr : STRING[80];
	a_dwConnectionHdl : ARRAY[1..c_diLFClntNum] OF DWORD;
	a_bNodeWr : ARRAY[1..c_diLFClntNum] OF BOOL;
	a_bNodeRd : ARRAY[1..c_diLFClntNum] OF BOOL;
	a_tyWriteHdls : ARRAY[1..c_diLFClntNum] OF tyOPCUAHdlList;
	a_tyReadHdls : ARRAY[1..c_diLFClntNum] OF tyOPCUAHdlList;
	eOPCUAStep : eLFOPCUAStep;
	fbConnect : fbOPCUAConnect;
	fbGetNodeHdlListWr : fbOPCUAGetNodeHdlList;
	fbGetNodeHdlListRd : fbOPCUAGetNodeHdlList;
	fbWriteList : fbOPCUAWriteList;
	fbDisconnect : fbOPCUADisconnect;
	fbReadList : fbOPCUAReadList;
	udiModuleNum : UDINT := 3801;
END_VAR
```

### Program Logical/LF/LFFollower (IEC, version 1.00.0) - 1.00.0 - NtHermes v5.00.0 , NtTCP v5.00.0 , NtMessage v5.00.0

#### Init.st - Change By Project
```iecst
(** 2020-08-06 **)
PROGRAM _INIT

	(* Always Change If Project Change *)

	//Physical Configuration
	bAutoUpdtData	:= TRUE;
	bInternalUse	:= FALSE;

	//Pass Address To Global Address For External Use
	//Action, State & Status
	p_LFFollowerStatus	:= ADR(eStatus);

	//Alarm
	p_LFFollowerAlmData		:= ADR(tyAlmData);
	p_LFFollowerInfoData	:= ADR(tyInfoData);
	p_LFFollowerInfoData1	:= ADR(tyInfoData1);

	//Output
	p_LFFollowerUSAllow			:= ADR(bUSAllow);
	p_LFFollowerDSAllow			:= ADR(bDSAllow);
	p_LFFollowerProdAccDataMnl	:= ADR(bProdAccDataMnl);
	p_LFFollowerProdUpdtDataMnl	:= ADR(bProdUpdtDataMnl);
	p_LFFollowerMagAccDataMnl	:= ADR(bMagAccDataMnl);
	p_LFFollowerTimeAct			:= ADR(eTimeAct);
	p_LFFollowerSetDT			:= ADR(tyLeaderToFollowerTag.dtTm);
	p_LFFollowerWaitRlsBrd		:= ADR(bWaitRlsBrd);
	p_LFFollowerUpdtProdRcp		:= ADR(tyUpdtProdRcp);
	p_LFFollowerLdrSeqCtrlInActive	:= ADR(bLeaderSeqCtrlInActive);

	(* Always Change If Project Change *)

END_PROGRAM
```

#### Act_InputConfig.st - Change By Project
```iecst
(** 2020-09-21 **)
ACTION Act_InputConfig:

	//Pass Data To Internal Use
	p_bUIProdAccData ACCESS p_UIProdAccData;
	p_bUIProdUpdtData ACCESS p_UIProdAccData;
	pa_tyProdRcpList ACCESS p_ProdRcpCurrList;
	p_tyCurrProdRcp ACCESS p_ProdRcpCurrRcp0;
	p_tyDispProdRcp ACCESS p_ProdRcpCurrRcp1;
	p_tyFollower ACCESS p_Follower2;

	//Link bPrep, bEn & bDis
	IF g_tyNtParamCurr.bProjLaneBPrep = FALSE THEN
		tylocalLFFollower.In.bDis	:= g_tyStartUp.bRun OR g_tyMcParamCurr.eUSCommA = McSetCommModHermes;
	ELSE
		tylocalLFFollower.In.bDis	:= g_tyStartUp.bRun OR g_tyMcParamCurr.eUSCommA = McSetCommModHermes OR g_tyMcParamCurr.eUSCommB = McSetCommModHermes;
	END_IF

	//Accept Condition with the relevant Information
	bFollowerInfo	:= tyFollowerToLeaderTag.bProdWidthErr OR bProdRcpErrNotExist OR bProdRcpErrWidthMismatch;

	bLeaderInfo		:= (tyLeaderToFollowerTag.bProdWidthUSWarn OR tyLeaderToFollowerTag.bProdWidthDSWarn
	OR ((tyLeaderToFollowerTag.bProdNameUSWarn OR tyLeaderToFollowerTag.bProdNameDSWarn)
	AND (g_tyNtParamCurr.bAWPrep = TRUE) AND (g_tyMcParamCurr.bAWDis = FALSE) AND (g_tyAW.eStat <>AWActGoWidthOff)));

	//Info Message
	IF bFollowerInfo THEN
		IF tyFollowerToLeaderTag.bProdWidthErr = TRUE OR bProdRcpErrWidthMismatch THEN

			p_sInfoMsg		:= 'Product Recipe Width Does Not Match';
			p_sInfoMsg		:= CONCAT(p_sInfoMsg , '$r$n');
			p_sInfoMsg		:= CONCAT(p_sInfoMsg , 'Check Product Width And');
			p_sInfoMsg		:= CONCAT(p_sInfoMsg , '$r$n');
			p_sInfoMsg		:= CONCAT(p_sInfoMsg , 'Leader Request Width');

		ELSIF bProdRcpErrNotExist THEN

			p_sInfoMsg		:= 'New Product Not Found';
			p_sInfoMsg		:= CONCAT(p_sInfoMsg , '$r$n');
			p_sInfoMsg		:= CONCAT(p_sInfoMsg , 'In Product Recipe List');
			p_sInfoMsg		:= CONCAT(p_sInfoMsg , '$r$n');
			p_sInfoMsg		:= CONCAT(p_sInfoMsg , 'Create New Product');
			p_sInfoMsg		:= CONCAT(p_sInfoMsg , '$r$n');
			p_sInfoMsg		:= CONCAT(p_sInfoMsg , 'In Product Setting');
		END_IF
	ELSE

		IF (tyLeaderToFollowerTag.sReqProdRcpNm<>p_tyCurrProdRcp.sRcpNm) AND (tyLeaderToFollowerTag.sReqProdRcpNm<>'')
			AND bLeaderInfo=FALSE THEN

			p_sInfoMsg		:= 'Leader Request New Recipe';
			p_sInfoMsg		:= CONCAT(p_sInfoMsg , '$r$n');
			p_sInfoMsg		:= CONCAT(p_sInfoMsg , 'Old Recipe Name : ');
			p_sInfoMsg		:= CONCAT(p_sInfoMsg , p_tyDispProdRcp.sRcpNm);
			p_sInfoMsg		:= CONCAT(p_sInfoMsg , '$r$n');
			p_sInfoMsg		:= CONCAT(p_sInfoMsg , 'Old Recipe Width : ');
			sWidthInUMTemp	:= DINT_TO_STRING(p_tyDispProdRcp.diWidthInUM / 1000);
			p_sInfoMsg		:= CONCAT(p_sInfoMsg , sWidthInUMTemp);
			p_sInfoMsg		:= CONCAT(p_sInfoMsg , '$r$n');
			p_sInfoMsg		:= CONCAT(p_sInfoMsg , 'New Recipe Name : ');
			p_sInfoMsg		:= CONCAT(p_sInfoMsg , tyLeaderToFollowerTag.sReqProdRcpNm);
			p_sInfoMsg		:= CONCAT(p_sInfoMsg , '$r$n');
			p_sInfoMsg		:= CONCAT(p_sInfoMsg , 'New Recipe Width : ');
			sWidthInUMTemp	:= DINT_TO_STRING(tyLeaderToFollowerTag.diReqProdRcpWidth / 1000);
			p_sInfoMsg		:= CONCAT(p_sInfoMsg , sWidthInUMTemp);

		ELSIF tyLeaderToFollowerTag.bProdNameUSWarn THEN
			p_sInfoMsg		:= 'US Machine Request New Recipe';
			p_sInfoMsg		:= CONCAT(p_sInfoMsg , '$r$n');
			p_sInfoMsg		:= CONCAT(p_sInfoMsg , 'Old Recipe Name : ');
			p_sInfoMsg		:= CONCAT(p_sInfoMsg , p_tyDispProdRcp.sRcpNm);
			p_sInfoMsg		:= CONCAT(p_sInfoMsg , '$r$n');
			p_sInfoMsg		:= CONCAT(p_sInfoMsg , 'Old Recipe Width : ');
			sWidthInUMTemp	:= DINT_TO_STRING(p_tyDispProdRcp.diWidthInUM / 1000);
			p_sInfoMsg		:= CONCAT(p_sInfoMsg , sWidthInUMTemp);
			p_sInfoMsg		:= CONCAT(p_sInfoMsg , '$r$n');
			p_sInfoMsg		:= CONCAT(p_sInfoMsg , 'New Recipe Name : ');
			p_sInfoMsg		:= CONCAT(p_sInfoMsg , tyLeaderToFollowerTag.sReqProdRcpNm);
			p_sInfoMsg		:= CONCAT(p_sInfoMsg , '$r$n');
			p_sInfoMsg		:= CONCAT(p_sInfoMsg , 'New Recipe Width : ');
			sWidthInUMTemp	:= DINT_TO_STRING(tyLeaderToFollowerTag.diReqProdRcpWidth / 1000);
			p_sInfoMsg		:= CONCAT(p_sInfoMsg , sWidthInUMTemp);

		ELSIF tyLeaderToFollowerTag.bProdNameDSWarn THEN
			p_sInfoMsg		:= 'Different Recipe';
			p_sInfoMsg		:= CONCAT(p_sInfoMsg , '$r$n');
			p_sInfoMsg		:= CONCAT(p_sInfoMsg , 'From DS Machine');
			p_sInfoMsg		:= CONCAT(p_sInfoMsg , '$r$n');
			p_sInfoMsg		:= CONCAT(p_sInfoMsg , 'Current Recipe Name : ');
			p_sInfoMsg		:= CONCAT(p_sInfoMsg , p_tyCurrProdRcp.sRcpNm);
			p_sInfoMsg		:= CONCAT(p_sInfoMsg , '$r$n');
			p_sInfoMsg		:= CONCAT(p_sInfoMsg , 'Current Recipe Width : ');
			sWidthInUMTemp	:= DINT_TO_STRING(p_tyCurrProdRcp.diWidthInUM2 / 1000);
			p_sInfoMsg		:= CONCAT(p_sInfoMsg , sWidthInUMTemp);

		ELSIF tyLeaderToFollowerTag.bProdWidthUSWarn THEN
			p_sInfoMsg		:= 'Product Recipe Width Does Not Match';
			p_sInfoMsg		:= CONCAT(p_sInfoMsg , '$r$n');
			p_sInfoMsg		:= CONCAT(p_sInfoMsg , 'Check Product Width And');
			p_sInfoMsg		:= CONCAT(p_sInfoMsg , '$r$n');
			p_sInfoMsg		:= CONCAT(p_sInfoMsg , 'Leader Request Width');

		ELSIF tyLeaderToFollowerTag.bProdWidthDSWarn THEN
			p_sInfoMsg		:= 'Same Recipe : ';
			p_sInfoMsg		:= CONCAT(p_sInfoMsg , p_tyDispProdRcp.sRcpNm);
			p_sInfoMsg		:= CONCAT(p_sInfoMsg , '$r$n');
			p_sInfoMsg		:= CONCAT(p_sInfoMsg , 'But Different Width');
			p_sInfoMsg		:= CONCAT(p_sInfoMsg , '$r$n');
			p_sInfoMsg		:= CONCAT(p_sInfoMsg , 'With DS Machine');
			p_sInfoMsg		:= CONCAT(p_sInfoMsg , '$r$n');
			p_sInfoMsg		:= CONCAT(p_sInfoMsg , 'Machine Outgoing Width : ');
			sWidthInUMTemp	:= DINT_TO_STRING(p_tyDispProdRcp.diWidthInUM2 / 1000);
			p_sInfoMsg		:= CONCAT(p_sInfoMsg , sWidthInUMTemp);

		END_IF
	END_IF

	//Accept New Recipe Condition (Before Loaded New Recipe)
	IF p_eLinkNtParamProjMag = ULMagDual OR p_eLinkNtParamProjMag = ULMagTriple  THEN
		p_bAccNewRcpCond	:= g_tyOps.bRun;  AND (g_tyPshrConv.bHvBrd = FALSE);
	END_IF

	//Update New Recipe Condition (After Loaded New Recipe)
	p_bUpdtNewRcpCond	:= TRUE;

	IF g_tyAlm.bErr THEN
		eCurrMachineStat := InError;
	ELSE
		IF g_tyAlm.bWarning THEN
			eCurrMachineStat := Warning;
		ELSE
			IF g_tyOps.bRun THEN
				eCurrMachineStat := Run;
			ELSE
				IF g_tyUIOut.bUIManualMod THEN
					eCurrMachineStat := Manual;
				ELSE
					eCurrMachineStat := Stop;
				END_IF
			END_IF
		END_IF
	END_IF

END_ACTION
```

#### Cyclic.st - Do Not Change!!!
```iecst
PROGRAM _CYCLIC

	IF bInitDone = FALSE THEN
		bInitDone	:= TRUE;
		Act_InitLocal;

	ELSIF bInitialDone = FALSE THEN
		IF g_tyStartUp.bNtSettingsLoadDone THEN
			bInitialDone	:= TRUE;
			Act_Initial;
		END_IF

	ELSE

		Act_InputConfig;

		IF (tylocalLFFollower.In.bPrep = TRUE) AND (tylocalLFFollower.In.bEn = TRUE) AND (tylocalLFFollower.In.bDis = FALSE) THEN
			Act_Background;

		ELSE
			Act_Main_Disable;
		END_IF

		Act_Alarm;

	END_IF

END_PROGRAM
```

#### Act_InitLocal.st - Do Not Change!!!
```iecst
ACTION Act_InitLocal:

	p_bUIProdAccData ACCESS ADR(bUIProdAccData);
	p_bUIProdUpdtData ACCESS ADR(bUIProdUpdtData);
	p_bUIMagAccData ACCESS ADR(bUIMagAccData);
	pa_tyProdRcpList ACCESS ADR(a_tyProdRcpList);
	p_tyCurrProdRcp ACCESS ADR(tyCurrProdRcp);
	p_tyDispProdRcp ACCESS ADR(tyDispProdRcp);
	p_sCurrMagRcpNm ACCESS ADR(sCurrMagRcpNm);
	p_bAccNewRcpCond ACCESS ADR(bAccNewRcpCond);
	p_bUpdtNewRcpCond ACCESS ADR(bUpdtNewRcpCond);
	p_bAutoUpdtData ACCESS ADR(bAutoUpdtData);
	p_sInfoMsg ACCESS ADR(sInfoMsg);
	p_bInternalUse ACCESS ADR(bInternalUse);
	p_tyInternalReqProdRcp ACCESS ADR(tyInternalReqProdRcp);
	p_bNewBrdEnteredCond ACCESS ADR(bNewBrdEnteredCond);
	p_bOldBrdExitedCond ACCESS ADR(bOldBrdExitedCond);
	p_bRlsBrd ACCESS ADR(bRlsBrd);
	p_bInternalReqProdRcpDiff ACCESS ADR(bInternalReqProdRcpDiff);
	p_bUpdtProdRcpDiff ACCESS ADR(bUpdtProdRcpDiff);
	p_bRlsBrdProdRcpDiff ACCESS ADR(bRlsBrdProdRcpDiff);

END_ACTION
```

#### Act_Initial.st - Do Not Change!!!
```iecst
ACTION Act_Initial:

	//Initial
	fbFollower.diWidthLimit	:= g_tyNtParamCurr.diLFWidthLimit;
	fbFollower(bEn := FALSE);

	fbOnlineChk.p_tyLeaderInfo		:= ADR(tyLeaderInfo);
	fbOnlineChk.tDlyTm				:= g_tyNtParamCurr.tLFFollowerOnlineChkDlyTm;
	fbOnlineChk(bEn := FALSE);

END_ACTION
```

#### Act_Background.st - Do Not Change!!!
```iecst
ACTION Act_Background:

	IF p_bInternalUse = TRUE THEN
		tyLeaderToFollowerTag.sReqProdRcpNm		:= p_tyInternalReqProdRcp.sRcpNm;

		IF g_tyNtParamCurr.bLFProdWidth2Prep THEN
			tyLeaderToFollowerTag.diReqProdRcpWidth	:= p_tyInternalReqProdRcp.diWidthInUM2;
		ELSE
			tyLeaderToFollowerTag.diReqProdRcpWidth	:= p_tyInternalReqProdRcp.diWidthInUM;
		END_IF
		tyLeaderToFollowerTag.sReqMagRcpNm		:= '';
		tyLeaderToFollowerTag.bMnlAccData		:= FALSE;
		tyLeaderToFollowerTag.bBypassMnlAccData	:= FALSE;
		tyLeaderToFollowerTag.bBlkDS			:= FALSE;
		tyLeaderToFollowerTag.bBlkUS			:= FALSE;
		tyLeaderToFollowerTag.bBypassWidthChk	:= TRUE;
		tyLeaderToFollowerTag.bSetTm			:= FALSE;
		tyLeaderToFollowerTag.dtTm				:= 0;
		tyLeaderToFollowerTag.uiTmZone			:= 0;
		tyLeaderToFollowerTag.usiRunTm			:= 0;
		tyLeaderToFollowerTag.bProdNameUSWarn	:= FALSE;
		tyLeaderToFollowerTag.bProdNameDSWarn	:= FALSE;
		tyLeaderToFollowerTag.bProdWidthUSWarn	:= FALSE;
		tyLeaderToFollowerTag.bProdWidthDSWarn	:= FALSE;
		tyLeaderToFollowerTag.bLeaderSeqCtrlInActive	:= FALSE;
	END_IF

	Act_Background_UpdtData;

	//FB
	fbFollower.tyLeaderToFollowerTag	:= tyLeaderToFollowerTag;
	fbFollower.sMcNm					:= g_tyMcParamCurr.sMcNm;
	fbFollower.sIPAddr					:= g_tyMcParamCurr.sIPAddr;
	fbFollower.bSectionLeader			:= g_tyMcParamCurr.bSectionLeader;
	fbFollower.sCurrProdRcpNm			:= p_tyCurrProdRcp.sRcpNm;
	fbFollower.diCurrProdWidthUS		:= p_tyCurrProdRcp.diWidthInUM;
	fbFollower.diCurrProdWidthDS		:= p_tyCurrProdRcp.diWidthInUM2;
	fbFollower.sCurrMagRcpNm			:= p_sCurrMagRcpNm;
	fbFollower.sUpdtLeaderProdRcpNm		:= p_tyFollower.tyUpdtProdRcp.sRcpNm;
	fbFollower.diUpdtLeaderProdWidthUS	:= p_tyFollower.tyUpdtProdRcp.diWidthInUM;
	fbFollower.diUpdtLeaderProdWidthDS	:= p_tyFollower.tyUpdtProdRcp.diWidthInUM2;
	fbFollower.sUpdtLeaderMagRcpNm		:= tylocalLFFollower.In.sMagRcpNm;
	fbFollower.bMnlAccDat				:= g_tyMcParamCurr.bMnlAccDat;
	fbFollower.bAWEn					:= (g_tyNtParamCurr.bAWPrep = TRUE) AND (g_tyMcParamCurr.bAWDis = FALSE);
	fbFollower.bUSWidthChkEn			:= g_tyNtParamCurr.bUSWidthChkPrep AND g_tyMcParamCurr.bUSWidthChkEn;
	fbFollower.bUSWidthChkSen			:= tylocalLFFollower.In.bUSWidthChkSen;
	fbFollower.bDSWidthChkEn			:= g_tyNtParamCurr.bDSWidthChkPrep AND g_tyMcParamCurr.bDSWidthChkEn;
	fbFollower.bDSWidthChkSen			:= tylocalLFFollower.In.bDSWidthChkSen;
	fbFollower.bProdWidthChk			:= g_tyNtParamCurr.bLFProdWidthChk;
	fbFollower.bProdRcpErr				:= bProdRcpErr;
	fbFollower.bMagRcpErr				:= bMagRcpErr;
	fbFollower.bSetTmErr				:= bSetTmErr;
	fbFollower.eCurrMachineStat			:= eCurrMachineStat;
	fbFollower.bProdChgOverActive		:= (g_tyAW.eStat = AWActGoWidthOff);
	fbFollower.bDBAOnWOAlign			:= g_tyMcParamCurr.bDBAOnWOAlign;

	fbFollower(bEn := TRUE);

	tyFollowerToLeaderTag	:= fbFollower.tyFollowerToLeaderTag;
	bProdAccDataReq			:= fbFollower.bProdAccDataReq OR (p_bInternalReqProdRcpDiff = TRUE) ;
	bMagAccDataReq			:= fbFollower.bMagAccDataReq;
	bAutoAccData			:= fbFollower.bAutoAccData;

	IF p_bInternalUse THEN
		bLeaderOnline			:= TRUE;
	ELSE
		bLeaderOnline			:= tyLeaderInfo.bOnline;
	END_IF

	IF bLeaderOnline=FALSE THEN
		bUSAllow				:= TRUE;
		bDSAllow				:= TRUE;
		bLeaderSeqCtrlInActive	:= FALSE;
	ELSE
		bUSAllow				:= fbFollower.bUSAllow AND (p_bInternalReqProdRcpDiff = FALSE);
		bDSAllow				:= fbFollower.bDSAllow;
		bLeaderSeqCtrlInActive	:= tyLeaderToFollowerTag.bLeaderSeqCtrlInActive;
	END_IF

	fbOnlineChk.tyLeaderToFollowerTag	:= tyLeaderToFollowerTag;
	fbOnlineChk(bEn := TRUE);

	Act_Background_AccData;
	Act_Background_ChkRlsBrd;

	//Set Time
	IF EDGEPOS(tyLeaderToFollowerTag.bSetTm) THEN
		bSetTm	:= TRUE;
	END_IF

	IF bSetTm = TRUE THEN
		eTimeAct	:= TimeActSetTime;

		IF (g_tyTime.eStat = TimeActSetTime) AND (g_tyTime.eMainStatus = Done) THEN
			eTimeAct		:= TimeActIdle;
			bSetTm			:= FALSE;
		ELSIF g_tyTime.eMainStatus = Error THEN
			eTimeAct		:= TimeActIdle;
			bSetTm			:= FALSE;
		END_IF
	END_IF

	bSetTmErr	:= g_tyTime.eMainStatus = Error;

	IF (eStatus = Error) AND bRstErr THEN
		eStatus		:= Idle;
		udiStatus	:= 0;
		bProdRcpErr	:= FALSE;
		bProdRcpErrNotExist	:= FALSE;
		bProdRcpErrWidthMismatch:= FALSE;
		bMagRcpErr	:= FALSE;
	END_IF

END_ACTION
```

#### Act_Background_ChkRlsBrd.st - Do Not Change!!!
```iecst
ACTION Act_Background_ChkRlsBrd:

	IF tyRlsBrdProdRcpNm.sRcpNm = '' THEN
		tyRlsBrdProdRcpNm	:= p_tyCurrProdRcp;

	ELSIF (tyRlsBrdProdRcpNm.sRcpNm <> p_tyCurrProdRcp.sRcpNm) OR (p_bRlsBrdProdRcpDiff = TRUE) THEN

		IF p_bNewBrdEnteredCond = TRUE THEN
			bNewBrdEntered	:= TRUE;
		END_IF

		IF p_bOldBrdExitedCond = TRUE THEN
			bOldBrdExited	:= TRUE;
		END_IF

		IF bNewBrdEntered AND bOldBrdExited THEN
			bWaitRlsBrd	:= TRUE;
		END_IF

		IF bWaitRlsBrd AND p_bRlsBrd THEN
			tyRlsBrdProdRcpNm	:= p_tyCurrProdRcp;
		END_IF

	ELSE
		bNewBrdEntered	:= FALSE;
		bOldBrdExited	:= FALSE;
		bWaitRlsBrd		:= FALSE;

	END_IF

END_ACTION
```

#### Act_Background_UpdtData.st - Do Not Change!!!
```iecst
ACTION Act_Background_UpdtData:

	//Update To Leader Recipe
	CASE usiProdUpdtDatStep OF
		0:
			//Update New Recipe Condition
			IF tyUpdtProdRcp.sRcpNm <> '' THEN
				IF (p_tyCurrProdRcp.sRcpNm <> tyUpdtProdRcp.sRcpNm) OR (p_bUpdtProdRcpDiff = TRUE) THEN
					IF p_bUpdtNewRcpCond = TRUE THEN
						usiProdUpdtDatStep	:= 1;
					END_IF
				END_IF
			ELSE
				tyUpdtProdRcp	:= p_tyCurrProdRcp;
			END_IF

		1:
			//Manual Update Data Check
			IF p_bAutoUpdtData = FALSE THEN
				bProdUpdtDataMnl	:= TRUE;

				IF p_bUIProdUpdtData = TRUE THEN
					bProdUpdtDataMnl	:= FALSE;
					usiProdUpdtDatStep	:= 2;
				END_IF
			ELSE
				bProdUpdtDataMnl	:= FALSE;
				usiProdUpdtDatStep	:= 2;
			END_IF

		2:
			//Update New Recipe
			tyUpdtProdRcp	:= p_tyCurrProdRcp;

			usiProdUpdtDatStep	:= 0;

	END_CASE

END_ACTION
```

#### Act_Background_AccData.st - Do Not Change!!!
```iecst
ACTION Act_Background_AccData:
	//Product Accept Data Request
	CASE usiProdAccDatStep OF
		0:
			//Check Error & Request Accept Data
			// If Product Name/Width Error, Check In Background To Update Data
			IF ((eStatus <> Error) AND (bProdAccDataReq = TRUE)) OR bProdRcpErr THEN
				sReqProdRcpNm		:= tyLeaderToFollowerTag.sReqProdRcpNm;
				diReqProdRcpWidth	:= tyLeaderToFollowerTag.diReqProdRcpWidth;
				usiProdAccDatStep	:= 1;
			END_IF

			IF bLeaderOnline=FALSE THEN
				tyInfoData.udiCode		:= 0;
				tyInfoData.eSeverity	:= AlmSeverityNA;

				bProdRcpErr 			:= FALSE;
				bProdRcpErrNotExist		:= FALSE;
				bProdRcpErrWidthMismatch:= FALSE;
			END_IF

		1:
			IF p_bInternalUse THEN
				usiProdAccDatStep	:= 2;
			ELSE
				//Check In List Of Recipe
				FOR i := 1 TO 2000 DO
					IF sReqProdRcpNm = '' THEN
						EXIT;
					ELSIF sReqProdRcpNm = pa_tyProdRcpList[i].sRcpNm  THEN
						EXIT;
					END_IF
				END_FOR

				IF sReqProdRcpNm = pa_tyProdRcpList[i].sRcpNm AND diReqProdRcpWidth <> pa_tyProdRcpList[i].diWidthInUM THEN
					//Width Mismatch
					bProdRcpErr := TRUE;
					bProdRcpErrWidthMismatch:= TRUE;
					bProdRcpErrNotExist		:= FALSE;
					usiProdAccDatStep	:= 0;
				ELSIF i > 2000 THEN
					//Recipe Not Exist
					bProdRcpErr := TRUE;
					bProdRcpErrNotExist	:= TRUE;
					bProdRcpErrWidthMismatch:= FALSE;
					usiProdAccDatStep	:= 0;
				ELSE
					bProdRcpErr := FALSE;
					bProdRcpErrNotExist	:= FALSE;
					bProdRcpErrWidthMismatch:= FALSE;
					usiProdAccDatStep	:= 2;
				END_IF

				//Info Message
				IF bLeaderOnline=FALSE THEN

					tyInfoData.udiCode		:= 0;
					tyInfoData.eSeverity	:= AlmSeverityNA;

					bProdRcpErr 			:= FALSE;
					bProdRcpErrNotExist		:= FALSE;
					bProdRcpErrWidthMismatch:= FALSE;
				ELSE
					IF p_bInternalUse = FALSE THEN
						IF bLeaderInfo OR bFollowerInfo THEN
//							tyInfoData.sProgNm		:= g_tyNtParamCurr.sLFFollowerProgNm;
							tyInfoData.udiCode		:= 10000;
							tyInfoData.eSeverity	:= AlmSeverityInfo;
							tyInfoData.sAlmMsg		:= p_sInfoMsg;
						ELSE
//							tyInfoData.sProgNm		:= '';
							tyInfoData.udiCode		:= 0;
							tyInfoData.eSeverity	:= AlmSeverityNA;

						END_IF
					ELSE
						IF p_sInfoMsg <> '' THEN
//							tyInfoData.sProgNm		:= g_tyNtParamCurr.sLFFollowerProgNm;
							tyInfoData.udiCode		:= 10000;
							tyInfoData.eSeverity	:= AlmSeverityInfo;
//							tyInfoData.sAlmMsg		:= p_sInfoMsg;
						ELSE
//							tyInfoData.sProgNm		:= '';
							tyInfoData.udiCode		:= 0;
							tyInfoData.eSeverity	:= AlmSeverityNA;
//							tyInfoData.sAlmMsg		:= '';
						END_IF
					END_IF
				END_IF
			END_IF

		2:
			//Manual Accept Data Check
			IF bProdAccDataReq = TRUE THEN
				IF bAutoAccData = FALSE THEN
					bProdAccDataMnl	:= TRUE;

					//Info Message
					IF bLeaderOnline=FALSE THEN
//						tyInfoData.sProgNm		:= '';
						tyInfoData.udiCode		:= 0;
						tyInfoData.eSeverity	:= AlmSeverityNA;
//						tyInfoData.sAlmMsg		:= '';
					ELSE
						IF p_sInfoMsg <> '' THEN
//							tyInfoData.sProgNm		:= g_tyNtParamCurr.sLFFollowerProgNm;
							tyInfoData.udiCode		:= 10000;
							tyInfoData.eSeverity	:= AlmSeverityInfo;
//							tyInfoData.sAlmMsg		:= p_sInfoMsg;
						ELSE
//							tyInfoData.sProgNm		:= '';
							tyInfoData.udiCode		:= 0;
							tyInfoData.eSeverity	:= AlmSeverityNA;
//							tyInfoData.sAlmMsg		:= '';
						END_IF
					END_IF

					IF p_bUIProdAccData = TRUE THEN
						p_bUIProdAccData := FALSE; //2023_07_26_Debug for Manual Accept Data automatically accept after product change many times
						bProdAccDataMnl		:= FALSE;
						usiProdAccDatStep	:= 3;
					END_IF
				ELSE
					bProdAccDataMnl		:= FALSE;
					p_bUIProdAccData := FALSE; //2023_07_26_Debug for Manual Accept Data automatically accept after product change many times
					usiProdAccDatStep	:= 3;
				END_IF
			ELSE
				bProdAccDataMnl		:= FALSE;
				usiProdAccDatStep	:= 6;
			END_IF

		3:
			//Accept New Recipe Condition
			IF bProdAccDataReq = TRUE THEN
				IF p_bAccNewRcpCond = TRUE THEN

					usiProdAccDatStep	:= 4;
				ELSE
					//Info Message
					IF bLeaderOnline=FALSE THEN
//						tyInfoData.sProgNm		:= '';
						tyInfoData.udiCode		:= 0;
						tyInfoData.eSeverity	:= AlmSeverityNA;
//						tyInfoData.sAlmMsg		:= '';
					ELSE
						IF p_sInfoMsg <> '' THEN
//							tyInfoData.sProgNm		:= g_tyNtParamCurr.sLFFollowerProgNm;
							tyInfoData.udiCode		:= 10000;
							tyInfoData.eSeverity	:= AlmSeverityInfo;
//							tyInfoData.sAlmMsg		:= p_sInfoMsg;
						ELSE
//							tyInfoData.sProgNm		:= '';
							tyInfoData.udiCode		:= 0;
							tyInfoData.eSeverity	:= AlmSeverityNA;
//							tyInfoData.sAlmMsg		:= '';
						END_IF
					END_IF
				END_IF
			ELSE
				usiProdAccDatStep	:= 6;
			END_IF

		4:
			//Accept New Recipe Name
			IF p_bInternalUse = TRUE THEN

				p_tyCurrProdRcp	:= p_tyInternalReqProdRcp;
				usiProdAccDatStep := 6;
			ELSE

				FOR i := 1 TO 2000 DO
					IF sReqProdRcpNm = '' THEN
						EXIT;
					ELSIF sReqProdRcpNm = pa_tyProdRcpList[i].sRcpNm THEN
						p_tyCurrProdRcp	:= pa_tyProdRcpList[i];
						EXIT;
					END_IF
				END_FOR

				IF i > 2000 THEN
					//Recipe Not Exist
					bProdRcpErr := TRUE;
					bProdRcpErrNotExist	:= TRUE;
				END_IF
				usiProdAccDatStep	:= 5;
			END_IF

		5:
			(* Add *)
			p_tyProdRcpCurrRcpWr 	:= p_tyCurrProdRcp;
			p_eLinkUIProdRcpAct 	:= ProdRcpActWriteCurrRcpParam;

			IF p_eProdRcpStat = ProdRcpActWriteCurrRcpParam AND p_eProdRcpStatus = Done THEN
				p_eLinkUIProdRcpAct := ProdRcpActIdle;
				usiProdAccDatStep := 6;
			END_IF

		6:
			//Clear Info Message
//			tyInfoData.sProgNm		:= '';
			tyInfoData.udiCode		:= 0;
			tyInfoData.eSeverity	:= AlmSeverityNA;
//			tyInfoData.sAlmMsg		:= '';

			usiProdAccDatStep	:= 0;

	END_CASE

END_ACTION
```

#### Act_Main_Disable.st - Do Not Change!!!
```iecst
ACTION Act_Main_Disable:

	bUSAllow			:= TRUE;
	bDSAllow			:= TRUE;
	bProdAccDataMnl		:= FALSE;
	bProdUpdtDataMnl	:= FALSE;
	bMagAccDataMnl		:= FALSE;
	bWaitRlsBrd			:= FALSE;

	usiProdAccDatStep		:= 0;
	usiProdUpdtDatStep		:= 0;
	tyInfoData.udiCode		:= 0;
	tyInfoData.eSeverity	:= AlmSeverityNA;

	usiMagAccDatStep		:= 0;
//	tyInfoData1.sProgNm		:= '';
	tyInfoData1.udiCode		:= 0;
	tyInfoData1.eSeverity	:= AlmSeverityNA;

	bSetTm		:= FALSE;

	eStatus		:= Idle;
	udiStatus	:= 0;
	bProdRcpErr	:= FALSE;
	bMagRcpErr	:= FALSE;
	bLeaderSeqCtrlInActive	:= FALSE;

	bProdRcpErrNotExist		:= FALSE;
	bProdRcpErrWidthMismatch:= FALSE;

END_ACTION
```

#### Act_Alarm.st - Do Not Change!!!
```iecst
ACTION Act_Alarm:

	IF g_tyRstErrOut.udiRstErr <> udiRstErrOld THEN
		bRstErr			:= TRUE;
		udiRstErrOld	:= g_tyRstErrOut.udiRstErr;
	ELSE
		bRstErr			:= FALSE;
	END_IF

	//Error
	IF EDGEPOS(eStatus = Error) THEN

		tylocalLFFollower.Out.tyAlmData.udiCode			:= udiStatus;
		tylocalLFFollower.Out.tyAlmData.eSeverity		:= AlmSeverityError;
		tylocalLFFollower.Out.tyAlmData.udiRunTime		:= tyAlmData.udiRunTime + 1;
		tylocalLFFollower.Out.tyAlmData.bAlm			:= TRUE;
		tylocalLFFollower.Out.tyAlmData.udiModuleNum	:= udiModuleNum;
		g_tyAlmProgNm.sLFFollowerProgNm					:= g_tyNtParamCurr.sLFFollowerProgNm;

	ELSIF bRstErr AND (tyAlmData.udiCode <> 0) THEN

		tylocalLFFollower.Out.tyAlmData.udiCode		:= 0;
		tylocalLFFollower.Out.tyAlmData.eSeverity	:= AlmSeverityNA;
		tylocalLFFollower.Out.tyAlmData.bAlm		:= FALSE;

	END_IF

END_ACTION
```

#### Local.var - Do Not Change!!!
```iecst
VAR
	tylocalLFFollower : tyLFFollower1;
END_VAR
(**)
VAR
	eStatus : eFBStatus := Idle;
	udiStatus : UDINT := 0;
END_VAR
(**)
(*Local Alarm*)
VAR
	tyAlmData : tyAlmDat;
	tyInfoData : tyAlmDat;
	tyInfoData1 : tyAlmDat;
END_VAR
(**)
(*Local Output*)
VAR
	bUSAllow : BOOL;
	bDSAllow : BOOL;
	bLeaderSeqCtrlInActive : BOOL;
	bProdAccDataMnl : BOOL;
	bProdUpdtDataMnl : BOOL;
	bMagAccDataMnl : BOOL;
	eTimeAct : eTimeAction;
	bWaitRlsBrd : BOOL;
	tyLeaderInfo : tyLFLeaderInfo;
	tyUpdtProdRcp : tyProdRcpParam;
END_VAR
(**)
VAR
	bUIProdAccData : BOOL;
	bUIProdUpdtData : BOOL;
	bUIMagAccData : BOOL;
	a_tyProdRcpList : ARRAY[1..c_udiProdRcpMax] OF tyProdRcpParam;
	tyDispProdRcp : tyProdRcpParam;
	tyCurrProdRcp : tyProdRcpParam;
	sCurrMagRcpNm : STRING[30];
	bAccNewRcpCond : BOOL;
	bUpdtNewRcpCond : BOOL;
	bAutoUpdtData : BOOL;
	sInfoMsg : STRING[200];
	bInternalUse : BOOL;
	tyInternalReqProdRcp : tyProdRcpParam;
	bNewBrdEnteredCond : BOOL;
	bOldBrdExitedCond : BOOL;
	bRlsBrd : BOOL;
	tyToLeaderProdRcp : tyProdRcpParam;
	bInternalReqProdRcpDiff : BOOL;
	bUpdtProdRcpDiff : BOOL;
	bRlsBrdProdRcpDiff : BOOL;
	sWidthInUMTemp : STRING[80];
END_VAR
(**)
(*Local*)
VAR
	bRstErr : BOOL;
	udiRstErrOld : UDINT;
	bInitDone : BOOL;
	bInitialDone : BOOL;
	bAutoAccData : BOOL;
	bProdRcpErr : BOOL;
	bMagRcpErr : BOOL;
	bSetTmErr : BOOL;
	bProdAccDataReq : BOOL;
	sReqProdRcpNm : STRING[254];
	diReqProdRcpWidth : DINT;
	bMagAccDataReq : BOOL;
	sReqMagRcpNm : STRING[30];
	usiProdAccDatStep : USINT;
	usiMagAccDatStep : USINT;
	usiProdUpdtDatStep : USINT;
	tyRlsBrdProdRcpNm : tyProdRcpParam;
	bNewBrdEntered : BOOL;
	bOldBrdExited : BOOL;
	i : INT;
	bSetTm : BOOL;
	fbOnlineChk : fbLFFollowerOnlineChk;
	fbFollower : fbLFFollower;
	tyLeaderToFollowerTag : tyLFLeaderToFollowerTag;
	tyFollowerToLeaderTag : tyLFFollowerToLeaderTag;
	eCurrMachineStat : eMachineStat;
	bLeaderOnline : BOOL;
	bLeaderInfo : BOOL;
	bFollowerInfo : BOOL;
	bProdRcpErrNotExist : BOOL;
	bProdRcpErrWidthMismatch : BOOL;
	p_bUIProdAccData : REFERENCE TO BOOL;
	p_bUIProdUpdtData : REFERENCE TO BOOL;
	p_bUIMagAccData : REFERENCE TO BOOL;
	pa_tyProdRcpList : REFERENCE TO ARRAY[1..c_udiProdRcpMax] OF tyProdRcpParam;
	p_tyCurrProdRcp : REFERENCE TO tyProdRcpParam;
	p_tyDispProdRcp : REFERENCE TO tyProdRcpParam;
	p_sCurrMagRcpNm : REFERENCE TO STRING[30];
	p_bAccNewRcpCond : REFERENCE TO BOOL;
	p_bUpdtNewRcpCond : REFERENCE TO BOOL;
	p_bAutoUpdtData : REFERENCE TO BOOL;
	p_sInfoMsg : REFERENCE TO STRING[200];
	p_bInternalUse : REFERENCE TO BOOL;
	p_tyInternalReqProdRcp : REFERENCE TO tyProdRcpParam;
	p_bNewBrdEnteredCond : REFERENCE TO BOOL;
	p_bOldBrdExitedCond : REFERENCE TO BOOL;
	p_bRlsBrd : REFERENCE TO BOOL;
	p_bInternalReqProdRcpDiff : REFERENCE TO BOOL;
	p_bUpdtProdRcpDiff : REFERENCE TO BOOL;
	p_bRlsBrdProdRcpDiff : REFERENCE TO BOOL;
	p_tyFollower : REFERENCE TO tyLFFollowerOut1;
	udiModuleNum : UDINT := 3901;
END_VAR
```

#### InputRef.var - not listed in the package file held
```iecst
(*2021-05-18*)
(**)
(*General*)
VAR
	p_udiRstErr : REFERENCE TO UDINT;
	p_bPrep : REFERENCE TO BOOL;
	p_bEn : REFERENCE TO BOOL;
	p_bDis : REFERENCE TO BOOL;
END_VAR
(**)
(*Configuration*)
VAR
	p_eAWStat : REFERENCE TO eAWAction;
	p_sIPAddr : REFERENCE TO STRING[15];
END_VAR
(**)
(*Input*)
VAR
	p_sMcNm : REFERENCE TO STRING[30];
	p_bAWPrep : REFERENCE TO BOOL;
	p_bAWDis : REFERENCE TO BOOL;
	p_bMnlAccData : REFERENCE TO BOOL;
	p_bSectionLeader : REFERENCE TO BOOL;
	p_sMagRcpNm : REFERENCE TO STRING[30];
	p_diWidthLimit : REFERENCE TO DINT;
	p_bWidth2Prep : REFERENCE TO BOOL;
	p_bUSWidthChkPrep : REFERENCE TO BOOL;
	p_bUSWidthChkEn : REFERENCE TO BOOL;
	p_bUSWidthChkSen : REFERENCE TO BOOL;
	p_bDSWidthChkPrep : REFERENCE TO BOOL;
	p_bDSWidthChkEn : REFERENCE TO BOOL;
	p_bDSWidthChkSen : REFERENCE TO BOOL;
	p_bProdWidthChk : REFERENCE TO BOOL;
	p_bUIProdAccData : REFERENCE TO BOOL;
	p_bUIProdUpdtData : REFERENCE TO BOOL;
	p_bUIMagAccData : REFERENCE TO BOOL;
	pa_tyProdRcpList : REFERENCE TO ARRAY[1..c_udiProdRcpMax] OF tyProdRcpParam;
	p_tyCurrProdRcp : REFERENCE TO tyProdRcpParam;
	p_tyDispProdRcp : REFERENCE TO tyProdRcpParam;
	p_sCurrMagRcpNm : REFERENCE TO STRING[30];
	p_eTimeStat : REFERENCE TO eTimeAction;
	p_eTimeStatus : REFERENCE TO eFBStatus;
	p_bAccNewRcpCond : REFERENCE TO BOOL;
	p_bUpdtNewRcpCond : REFERENCE TO BOOL;
	p_bAutoUpdtData : REFERENCE TO BOOL;
	p_sInfoMsg : REFERENCE TO STRING[200];
	p_bInternalUse : REFERENCE TO BOOL;
	p_tyInternalReqProdRcp : REFERENCE TO tyProdRcpParam;
	p_bNewBrdEnteredCond : REFERENCE TO BOOL;
	p_bOldBrdExitedCond : REFERENCE TO BOOL;
	p_bRlsBrd : REFERENCE TO BOOL;
	p_tyToLeaderProdRcp : REFERENCE TO tyProdRcpParam;
	p_bInternalReqProdRcpDiff : REFERENCE TO BOOL;
	p_bUpdtProdRcpDiff : REFERENCE TO BOOL;
	p_bRlsBrdProdRcpDiff : REFERENCE TO BOOL;
	p_sProgNm : REFERENCE TO STRING[254];
	p_bNtSettingsLoadDone : REFERENCE TO BOOL;
	p_tOnlineChkDlyTm : REFERENCE TO TIME;
	p_bManual : REFERENCE TO BOOL;
	p_bErr : REFERENCE TO BOOL;
	p_bWarning : REFERENCE TO BOOL;
	p_bOps : REFERENCE TO BOOL;
	p_bStandby : REFERENCE TO BOOL;
	p_bDBAOnWOAlign : REFERENCE TO BOOL;
END_VAR
```

#### InputRef_Link.var - not listed in the package file held
```iecst
(*2019-05-07*)
(**)
VAR
	p_bLinkOpsRun : REFERENCE TO BOOL;
	p_bLinkStartupRun : REFERENCE TO BOOL;
	p_eLinkMcParamUSCommMod : REFERENCE TO eMcSetCommMod;
	p_bLinkAWWidthPosDiff : REFERENCE TO BOOL;
	p_bLinkConvBffrLastProduct : REFERENCE TO BOOL;
	p_bLinkBufferLastProductUnload : REFERENCE TO BOOL;
	p_tyLinkBufferBffrStat : REFERENCE TO tyBffrStat;
	p_bLinkNtParamProjLaneBPrep : REFERENCE TO BOOL;
	p_eLinkMcParamUSACommMod : REFERENCE TO eMcSetCommMod;
	p_eLinkMcParamUSBCommMod : REFERENCE TO eMcSetCommMod;
	p_eLinkNtParamProjMag : REFERENCE TO eULMag;
	p_bLinkPshrConvHvBrd : REFERENCE TO BOOL;
	p_bLinkBffr1MagRemoved : REFERENCE TO BOOL;
	p_bLinkBffr2MagRemoved : REFERENCE TO BOOL;
	p_bLinkBffr3MagRemoved : REFERENCE TO BOOL;
END_VAR
(**)
(**)
VAR
	sWidthInUMTemp : STRING[80];
END_VAR
VAR
	p_eLinkUIProdRcpAct : REFERENCE TO eProdRcpAction;
	p_eProdRcpStat : REFERENCE TO eProdRcpAction;
	p_eProdRcpStatus : REFERENCE TO eFBStatus;
	p_tyProdRcpCurrRcpWr : REFERENCE TO tyProdRcpParam;
END_VAR
```

#### Act_InitGlobal.st - not listed in the package file held
```iecst
(** 2020-09-21 **)
ACTION Act_InitGlobal:

	(* Always Change If Project Change *)

	//Pass Data To Link
	p_bLinkOpsRun ACCESS p_OpsRun;
	p_bLinkStartupRun ACCESS p_StartupRun;

	p_bLinkNtParamProjLaneBPrep ACCESS p_NtParamProjLaneBPrep;
	p_eLinkMcParamUSACommMod ACCESS p_McParamUSCommAMod;
	p_eLinkMcParamUSBCommMod ACCESS p_McParamUSCommBMod;

	p_eLinkNtParamProjMag ACCESS p_NtParamProjMag;
	p_bLinkPshrConvHvBrd ACCESS p_PshrConvHvBrd;
	p_bLinkBffr1MagRemoved ACCESS p_Buffer1MagRemoved;
	p_bLinkBffr2MagRemoved ACCESS p_Buffer2MagRemoved;
	p_bLinkBffr3MagRemoved ACCESS p_Buffer3MagRemoved;

	//Pass Data To Internal Use
	p_udiRstErr ACCESS p_RstErrReset;
	p_bPrep ACCESS p_NtParamLFPrep;
	p_bEn ACCESS p_McParamLFEn;
	p_sIPAddr ACCESS p_HWInfoIPAddr;
	p_sMcNm ACCESS p_McParamMcNm;
	p_bAWPrep ACCESS p_NtParamAWPrep;
	p_bAWDis ACCESS p_McParamAWDis;
	p_bMnlAccData ACCESS p_McParamMnlAccDat;
	p_bSectionLeader ACCESS p_McParamSectionLeader;
	p_diWidthLimit ACCESS p_NtParamLFWidthLimit;
	p_bProdWidthChk ACCESS p_NtParamLFProdWidthChk;
	p_bUIProdAccData ACCESS p_UIProdAccData;
	p_bUIMagAccData ACCESS p_UIMagAccData;
	pa_tyProdRcpList ACCESS p_ProdRcpCurrList;
	p_tyCurrProdRcp ACCESS p_ProdRcpCurrRcp0;
	p_tyDispProdRcp ACCESS p_ProdRcpCurrRcp1;
//	p_sCurrMagRcpNm ACCESS ADR(p_tyCurrMagRcp.sRcpNm);
	p_eTimeStat ACCESS p_TimeStat;
	p_eTimeStatus ACCESS p_TimeStatus;
	//	p_tyToLeaderProdRcp ACCESS p_Follower2UpdtProdRcp;	//Assign With Conveyor Last Zone (To Leader Completion Update)
	p_tyToLeaderProdRcp ACCESS p_Follower1UpdtProdRcp;	//Assign With Conveyor Last Zone (To Leader Completion Update)
	p_sProgNm ACCESS p_NtParamLFFollowerProgNm;
	p_bNtSettingsLoadDone ACCESS p_StartupNtSettingsLoadDone;

	p_tOnlineChkDlyTm ACCESS p_NtParamLFFllowerOnlineChkDlyTm;
	p_bManual ACCESS p_UIUIMnlMod;
	p_bErr ACCESS p_AlarmErr;
	p_bOps ACCESS p_OpsStatusRun;
	p_bStandby ACCESS p_OpsStatusStop;
	p_bWarning ACCESS p_AlarmWarning;
	p_eAWStat ACCESS p_AWOpenStat;
	p_bWidth2Prep ACCESS p_NtParamLFWidth2Prep;

	p_eProdRcpStat ACCESS p_ProdRcpStat; //add
	p_eProdRcpStatus ACCESS p_ProdRcpStatus; //add
	p_eLinkUIProdRcpAct ACCESS p_UIProdRcpAct; //add
	p_tyProdRcpCurrRcpWr ACCESS p_UIProdRcpCurrRcpWr; //add
	p_bDBAOnWOAlign ACCESS p_McParamDBAOnWOAlign;
	(* Always Change If Project Change *)

END_ACTION
```

#### Act_Link.st - not listed in the package file held
```iecst
(** 2021-05-18 **)
ACTION Act_Link:

	//ProdRcp
	bFollowerInfo	:= tyFollowerToLeaderTag.bProdWidthErr OR bProdRcpErrNotExist OR bProdRcpErrWidthMismatch;

	bLeaderInfo		:= (tyLeaderToFollowerTag.bProdWidthUSWarn OR tyLeaderToFollowerTag.bProdWidthDSWarn
	OR ((tyLeaderToFollowerTag.bProdNameUSWarn OR tyLeaderToFollowerTag.bProdNameDSWarn)
	AND (p_bAWPrep = TRUE) AND (p_bAWDis = FALSE) AND (p_eAWStat<>AWActGoWidthOff)));

	//Info Message
	IF bFollowerInfo THEN
		IF tyFollowerToLeaderTag.bProdWidthErr = TRUE OR bProdRcpErrWidthMismatch THEN

			p_sInfoMsg		:= 'Product Recipe Width Does Not Match';
			p_sInfoMsg		:= CONCAT(p_sInfoMsg , '$r$n');
			p_sInfoMsg		:= CONCAT(p_sInfoMsg , 'Check Product Width And');
			p_sInfoMsg		:= CONCAT(p_sInfoMsg , '$r$n');
			p_sInfoMsg		:= CONCAT(p_sInfoMsg , 'Leader Request Width');

		ELSIF bProdRcpErrNotExist THEN

			p_sInfoMsg		:= 'New Product Not Found';
			p_sInfoMsg		:= CONCAT(p_sInfoMsg , '$r$n');
			p_sInfoMsg		:= CONCAT(p_sInfoMsg , 'In Product Recipe List');
			p_sInfoMsg		:= CONCAT(p_sInfoMsg , '$r$n');
			p_sInfoMsg		:= CONCAT(p_sInfoMsg , 'Create New Product');
			p_sInfoMsg		:= CONCAT(p_sInfoMsg , '$r$n');
			p_sInfoMsg		:= CONCAT(p_sInfoMsg , 'In Product Setting');
		END_IF
	ELSE

		IF (tyLeaderToFollowerTag.sReqProdRcpNm<>p_tyCurrProdRcp.sRcpNm) AND (tyLeaderToFollowerTag.sReqProdRcpNm<>'')
			AND bLeaderInfo=FALSE THEN

			p_sInfoMsg		:= 'Leader Request New Recipe';
			p_sInfoMsg		:= CONCAT(p_sInfoMsg , '$r$n');
			p_sInfoMsg		:= CONCAT(p_sInfoMsg , 'Old Recipe Name : ');
			p_sInfoMsg		:= CONCAT(p_sInfoMsg , p_tyDispProdRcp.sRcpNm);
			p_sInfoMsg		:= CONCAT(p_sInfoMsg , '$r$n');
			p_sInfoMsg		:= CONCAT(p_sInfoMsg , 'Old Recipe Width : ');
			sWidthInUMTemp	:= DINT_TO_STRING(p_tyDispProdRcp.diWidthInUM / 1000);
			p_sInfoMsg		:= CONCAT(p_sInfoMsg , sWidthInUMTemp);
			p_sInfoMsg		:= CONCAT(p_sInfoMsg , '$r$n');
			p_sInfoMsg		:= CONCAT(p_sInfoMsg , 'New Recipe Name : ');
			p_sInfoMsg		:= CONCAT(p_sInfoMsg , tyLeaderToFollowerTag.sReqProdRcpNm);
			p_sInfoMsg		:= CONCAT(p_sInfoMsg , '$r$n');
			p_sInfoMsg		:= CONCAT(p_sInfoMsg , 'New Recipe Width : ');
			sWidthInUMTemp	:= DINT_TO_STRING(tyLeaderToFollowerTag.diReqProdRcpWidth / 1000);
			p_sInfoMsg		:= CONCAT(p_sInfoMsg , sWidthInUMTemp);

		ELSIF tyLeaderToFollowerTag.bProdNameUSWarn THEN
			p_sInfoMsg		:= 'US Machine Request New Recipe';
			p_sInfoMsg		:= CONCAT(p_sInfoMsg , '$r$n');
			p_sInfoMsg		:= CONCAT(p_sInfoMsg , 'Old Recipe Name : ');
			p_sInfoMsg		:= CONCAT(p_sInfoMsg , p_tyDispProdRcp.sRcpNm);
			p_sInfoMsg		:= CONCAT(p_sInfoMsg , '$r$n');
			p_sInfoMsg		:= CONCAT(p_sInfoMsg , 'Old Recipe Width : ');
			sWidthInUMTemp	:= DINT_TO_STRING(p_tyDispProdRcp.diWidthInUM / 1000); //Modify 18052021
			p_sInfoMsg		:= CONCAT(p_sInfoMsg , sWidthInUMTemp);
			p_sInfoMsg		:= CONCAT(p_sInfoMsg , '$r$n');
			p_sInfoMsg		:= CONCAT(p_sInfoMsg , 'New Recipe Name : ');
			p_sInfoMsg		:= CONCAT(p_sInfoMsg , tyLeaderToFollowerTag.sReqProdRcpNm);
			p_sInfoMsg		:= CONCAT(p_sInfoMsg , '$r$n');
			p_sInfoMsg		:= CONCAT(p_sInfoMsg , 'New Recipe Width : ');
			sWidthInUMTemp	:= DINT_TO_STRING(tyLeaderToFollowerTag.diReqProdRcpWidth / 1000);
			p_sInfoMsg		:= CONCAT(p_sInfoMsg , sWidthInUMTemp);

		ELSIF tyLeaderToFollowerTag.bProdNameDSWarn THEN
			p_sInfoMsg		:= 'Different Recipe';
			p_sInfoMsg		:= CONCAT(p_sInfoMsg , '$r$n');
			p_sInfoMsg		:= CONCAT(p_sInfoMsg , 'From DS Machine');
			p_sInfoMsg		:= CONCAT(p_sInfoMsg , '$r$n');
			p_sInfoMsg		:= CONCAT(p_sInfoMsg , 'Current Recipe Name : ');
			p_sInfoMsg		:= CONCAT(p_sInfoMsg , p_tyCurrProdRcp.sRcpNm);
			p_sInfoMsg		:= CONCAT(p_sInfoMsg , '$r$n');
			p_sInfoMsg		:= CONCAT(p_sInfoMsg , 'Current Recipe Width : ');
			sWidthInUMTemp	:= DINT_TO_STRING(p_tyCurrProdRcp.diWidthInUM2 / 1000);
			p_sInfoMsg		:= CONCAT(p_sInfoMsg , sWidthInUMTemp);

		ELSIF tyLeaderToFollowerTag.bProdWidthUSWarn THEN
			p_sInfoMsg		:= 'Product Recipe Width Does Not Match';
			p_sInfoMsg		:= CONCAT(p_sInfoMsg , '$r$n');
			p_sInfoMsg		:= CONCAT(p_sInfoMsg , 'Check Product Width And');
			p_sInfoMsg		:= CONCAT(p_sInfoMsg , '$r$n');
			p_sInfoMsg		:= CONCAT(p_sInfoMsg , 'Leader Request Width');

		ELSIF tyLeaderToFollowerTag.bProdWidthDSWarn THEN
			p_sInfoMsg		:= 'Same Recipe : ';
			p_sInfoMsg		:= CONCAT(p_sInfoMsg , p_tyDispProdRcp.sRcpNm);
			p_sInfoMsg		:= CONCAT(p_sInfoMsg , '$r$n');
			p_sInfoMsg		:= CONCAT(p_sInfoMsg , 'But Different Width');
			p_sInfoMsg		:= CONCAT(p_sInfoMsg , '$r$n');
			p_sInfoMsg		:= CONCAT(p_sInfoMsg , 'With DS Machine');
			p_sInfoMsg		:= CONCAT(p_sInfoMsg , '$r$n');
			p_sInfoMsg		:= CONCAT(p_sInfoMsg , 'Machine Outgoing Width : ');
			sWidthInUMTemp	:= DINT_TO_STRING(p_tyDispProdRcp.diWidthInUM2 / 1000);
			p_sInfoMsg		:= CONCAT(p_sInfoMsg , sWidthInUMTemp);

		END_IF
	END_IF

	//Accept New Recipe Condition (Before Loaded New Recipe)
	IF p_eLinkNtParamProjMag = ULMagDual OR p_eLinkNtParamProjMag = ULMagTriple  THEN
		p_bAccNewRcpCond	:= (p_bLinkOpsRun = TRUE)  AND (p_bLinkPshrConvHvBrd = FALSE);
	END_IF

	//Update New Recipe Condition (After Loaded New Recipe)
	p_bUpdtNewRcpCond	:= TRUE;

	//Recipe Different
	//p_bInternalReqProdRcpDiff	:= memcmp(ADR(p_tyCurrProdRcp) , ADR(p_tyInternalReqProdRcp) , SIZEOF(p_tyCurrProdRcp)) <> 0;
	//p_bUpdtProdRcpDiff			:= memcmp(ADR(p_tyCurrProdRcp) , ADR(tyUpdtProdRcp) , SIZEOF(p_tyCurrProdRcp)) <> 0;
	//p_bRlsBrdProdRcpDiff		:= memcmp(ADR(p_tyCurrProdRcp) , ADR(tyRlsBrdProdRcpNm) , SIZEOF(p_tyCurrProdRcp)) <> 0;

	IF p_bErr THEN
		eCurrMachineStat := InError;
	ELSE
		IF p_bWarning THEN
			eCurrMachineStat := Warning;
		ELSE
			IF p_bOps THEN
				eCurrMachineStat := Run;
			ELSE
				IF p_bManual THEN
					eCurrMachineStat := Manual;
				ELSE
					eCurrMachineStat := Stop;
				END_IF
			END_IF
		END_IF
	END_IF

END_ACTION
```

#### Act_LinkEn.st - not listed in the package file held
```iecst
(** 2019-04-26 **)
ACTION Act_LinkEn:

	//Link bPrep, bEn & bDis
	IF p_bLinkNtParamProjLaneBPrep = FALSE THEN
		p_bDis	:= (p_bLinkStartupRun = TRUE) OR (p_eLinkMcParamUSACommMod = McSetCommModHermes);
	ELSE
		p_bDis	:= (p_bLinkStartupRun = TRUE) OR (p_eLinkMcParamUSACommMod = McSetCommModHermes) OR (p_eLinkMcParamUSBCommMod = McSetCommModHermes);
	END_IF

END_ACTION
```

### Program Logical/LF/Follower1 (IEC) - 1.00.0 - NtHermes v5.00.0 , NtTCP v5.00.0 , NtMessage v5.00.0

#### InputRef.var
```iecst
(*2020-08-06*)
(**)
(*General*)
VAR
	p_udiRstErr : REFERENCE TO UDINT;
	p_bPrep : REFERENCE TO BOOL;
	p_bEn : REFERENCE TO BOOL;
	p_bDis : REFERENCE TO BOOL;
END_VAR
(**)
(*Configuration*)
VAR
	p_eAWStat : REFERENCE TO eAWAction;
	p_sIPAddr : REFERENCE TO STRING[15];
END_VAR
(**)
(*Input*)
VAR
	p_sMcNm : REFERENCE TO STRING[30];
	p_bAWPrep : REFERENCE TO BOOL;
	p_bAWDis : REFERENCE TO BOOL;
	p_bMnlAccData : REFERENCE TO BOOL;
	p_bSectionLeader : REFERENCE TO BOOL;
	p_sMagRcpNm : REFERENCE TO STRING[30];
	p_diWidthLimit : REFERENCE TO DINT;
	p_bWidth2Prep : REFERENCE TO BOOL;
	p_bNtParamAutoRcpPrep : REFERENCE TO BOOL;
	p_bMcParamAutoRcpDis : REFERENCE TO BOOL;
	p_eNtParamAutoRcpPrecededBy : REFERENCE TO eAutoRcpPreceded;
	p_bUSWidthChkPrep : REFERENCE TO BOOL;
	p_bUSWidthChkEn : REFERENCE TO BOOL;
	p_bUSWidthChkSen : REFERENCE TO BOOL;
	p_bDSWidthChkPrep : REFERENCE TO BOOL;
	p_bDSWidthChkEn : REFERENCE TO BOOL;
	p_bDSWidthChkSen : REFERENCE TO BOOL;
	p_bProdWidthChk : REFERENCE TO BOOL;
	p_bUIProdAccData : REFERENCE TO BOOL;
	p_bUIProdUpdtData : REFERENCE TO BOOL;
	p_bUIMagAccData : REFERENCE TO BOOL;
	pa_tyProdRcpList : REFERENCE TO ARRAY[1..c_udiProdRcpMax] OF tyProdRcpParam;
	p_tyCurrProdRcp : REFERENCE TO tyProdRcpParam;
	p_sCurrMagRcpNm : REFERENCE TO STRING[30];
	p_eTimeStat : REFERENCE TO eTimeAction;
	p_eTimeStatus : REFERENCE TO eFBStatus;
	p_bAccNewRcpCond : REFERENCE TO BOOL;
	p_bUpdtNewRcpCond : REFERENCE TO BOOL;
	p_bAutoUpdtData : REFERENCE TO BOOL;
	p_sInfoMsg : REFERENCE TO STRING[200];
	p_bInternalUse : REFERENCE TO BOOL;
	p_tyInternalReqProdRcp : REFERENCE TO tyProdRcpParam;
	p_bNewBrdEnteredCond : REFERENCE TO BOOL;
	p_bOldBrdExitedCond : REFERENCE TO BOOL;
	p_bRlsBrd : REFERENCE TO BOOL;
	p_tyToLeaderProdRcp : REFERENCE TO tyProdRcpParam;
	p_bInternalReqProdRcpDiff : REFERENCE TO BOOL;
	p_bUpdtProdRcpDiff : REFERENCE TO BOOL;
	p_bRlsBrdProdRcpDiff : REFERENCE TO BOOL;
	p_sProgNm : REFERENCE TO STRING[15];
	p_bNtSettingsLoadDone : REFERENCE TO BOOL;
	p_tOnlineChkDlyTm : REFERENCE TO TIME;
	p_bManual : REFERENCE TO BOOL;
	p_bErr : REFERENCE TO BOOL;
	p_bWarning : REFERENCE TO BOOL;
	p_bOps : REFERENCE TO BOOL;
	p_bStandby : REFERENCE TO BOOL;
	p_bDBAOnWOAlign : REFERENCE TO BOOL;
END_VAR
```

#### InputRef_Link.var
```iecst
(*2019-05-07*)
(**)
VAR
	p_bLinkOpsRun : REFERENCE TO BOOL;
	p_bLinkStartupRun : REFERENCE TO BOOL;
END_VAR
(**)
VAR
	p_bLinkPshrConvHvBrd : REFERENCE TO BOOL;
	p_bLinkOpsTravLifULInitDone : REFERENCE TO BOOL;
	p_eLinkUIProdRcpAct : REFERENCE TO eProdRcpAction;
	p_eProdRcpStat : REFERENCE TO eProdRcpAction;
	p_eProdRcpStatus : REFERENCE TO eFBStatus;
	p_tyProdRcpCurrRcpWr : REFERENCE TO tyProdRcpParam;
END_VAR
```

#### Local.var
```iecst
VAR
	tylocalFollower : tyLFFollower1;
END_VAR
(**)
VAR
	udiStatus : UDINT := 0;
END_VAR
(**)
(*Local Alarm*)
VAR
	tyAlmData : tyAlmDat;
	tyInfoData : tyAlmDat;
	tyInfoData1 : tyAlmDat;
END_VAR
(**)
VAR
	sMagRcpNm : STRING[30];
	bUIProdAccData : BOOL;
	bUIProdUpdtData : BOOL;
	bUIMagAccData : BOOL;
	a_tyProdRcpList : ARRAY[1..c_udiProdRcpMax] OF tyProdRcpParam;
	tyDispProdRcp : tyProdRcpParam;
	tyCurrProdRcp : tyProdRcpParam;
	sCurrMagRcpNm : STRING[30];
	bAccNewRcpCond : BOOL;
	bUpdtNewRcpCond : BOOL;
	bAutoUpdtData : BOOL;
	sInfoMsg : STRING[200];
	bInternalUse : BOOL;
	tyInternalReqProdRcp : tyProdRcpParam;
	bNewBrdEnteredCond : BOOL;
	bOldBrdExitedCond : BOOL;
	bRlsBrd : BOOL;
	tyToLeaderProdRcp : tyProdRcpParam;
	bInternalReqProdRcpDiff : BOOL;
	bUpdtProdRcpDiff : BOOL;
	bRlsBrdProdRcpDiff : BOOL;
	sWidthInUMTemp : STRING[80];
END_VAR
(**)
(*Local*)
VAR
	bRstErr : BOOL;
	udiRstErrOld : UDINT;
	bInitDone : BOOL;
	bInitialDone : BOOL;
	bAutoAccData : BOOL;
	bProdRcpErr : BOOL;
	bMagRcpErr : BOOL;
	bSetTmErr : BOOL;
	bProdAccDataReq : BOOL;
	sReqProdRcpNm : STRING[254];
	diReqProdRcpWidth : DINT;
	bMagAccDataReq : BOOL;
	sReqMagRcpNm : STRING[30];
	usiProdAccDatStep : USINT;
	usiMagAccDatStep : USINT;
	usiProdUpdtDatStep : USINT;
	tyRlsBrdProdRcpNm : tyProdRcpParam;
	bNewBrdEntered : BOOL;
	bOldBrdExited : BOOL;
	i : INT;
	bSetTm : BOOL;
	fbOnlineChk : fbLFFollowerOnlineChk;
	fbFollower : fbLFFollower;
	tyLeaderToFollowerTag : tyLFLeaderToFollowerTag;
	tyFollowerToLeaderTag : tyLFFollowerToLeaderTag;
	eCurrMachineStat : eMachineStat;
	bLeaderOnline : BOOL;
	bLeaderInfo : BOOL;
	bFollowerInfo : BOOL;
	bProdRcpErrNotExist : BOOL;
	bProdRcpErrWidthMismatch : BOOL;
	tyFollower : {REDUND_UNREPLICABLE} tyLFFollowerOut1;
END_VAR
(**)
VAR
	p_sMagRcpNm : REFERENCE TO STRING[30];
	p_bUIProdAccData : REFERENCE TO BOOL;
	p_bUIProdUpdtData : REFERENCE TO BOOL;
	p_bUIMagAccData : REFERENCE TO BOOL;
	pa_tyProdRcpList : REFERENCE TO ARRAY[1..c_udiProdRcpMax] OF tyProdRcpParam;
	p_tyCurrProdRcp : REFERENCE TO tyProdRcpParam;
	p_tyDispProdRcp : REFERENCE TO tyProdRcpParam;
	p_sCurrMagRcpNm : REFERENCE TO STRING[30];
	p_bAccNewRcpCond : REFERENCE TO BOOL;
	p_bUpdtNewRcpCond : REFERENCE TO BOOL;
	p_bAutoUpdtData : REFERENCE TO BOOL;
	p_sInfoMsg : REFERENCE TO STRING[200];
	p_bInternalUse : REFERENCE TO BOOL;
	p_tyInternalReqProdRcp : REFERENCE TO tyProdRcpParam;
	p_bNewBrdEnteredCond : REFERENCE TO BOOL;
	p_bOldBrdExitedCond : REFERENCE TO BOOL;
	p_bRlsBrd : REFERENCE TO BOOL;
	p_bInternalReqProdRcpDiff : REFERENCE TO BOOL;
	p_bUpdtProdRcpDiff : REFERENCE TO BOOL;
	p_bRlsBrdProdRcpDiff : REFERENCE TO BOOL;
	p_tyFollower : REFERENCE TO tyLFFollowerOut1;
	udiModuleNum : UDINT := 3901;
END_VAR
```

#### Act_Alarm.st
```iecst
ACTION Act_Alarm:

	IF g_tyRstErrOut.udiRstErr <> udiRstErrOld THEN
		bRstErr			:= TRUE;
		udiRstErrOld	:= g_tyRstErrOut.udiRstErr;
	ELSE
		bRstErr			:= FALSE;
	END_IF

	//Error
	IF EDGEPOS(tylocalFollower.Out.eStatus = Error) THEN

		tylocalFollower.Out.tyAlmData.udiCode		:= udiStatus;
		tylocalFollower.Out.tyAlmData.eSeverity		:= AlmSeverityError;
		tylocalFollower.Out.tyAlmData.udiRunTime	:= tyAlmData.udiRunTime + 1;
		tylocalFollower.Out.tyAlmData.bAlm			:= TRUE;
		tylocalFollower.Out.tyAlmData.udiModuleNum	:= udiModuleNum;
		g_tyAlmProgNm.sLFFollowerProgNm				 := g_tyNtParamCurr.sFollower1ProgNm;

	ELSIF bRstErr AND (tylocalFollower.Out.tyAlmData.udiCode <> 0) THEN

		tylocalFollower.Out.tyAlmData.udiCode	:= 0;
		tylocalFollower.Out.tyAlmData.eSeverity	:= AlmSeverityNA;
		tylocalFollower.Out.tyAlmData.bAlm		:= FALSE;

	END_IF

END_ACTION
```

#### Act_Background.st
```iecst
ACTION Act_Background:

	IF p_bInternalUse = TRUE THEN
		tyLeaderToFollowerTag.sReqProdRcpNm		:= p_tyInternalReqProdRcp.sRcpNm;

		IF g_tyNtParamCurr.bLFProdWidth2Prep THEN
			tyLeaderToFollowerTag.diReqProdRcpWidth	:= p_tyInternalReqProdRcp.diWidthInUM2;
		ELSE
			tyLeaderToFollowerTag.diReqProdRcpWidth	:= p_tyInternalReqProdRcp.diWidthInUM;
		END_IF
		tyLeaderToFollowerTag.sReqMagRcpNm		:= '';
		tyLeaderToFollowerTag.bMnlAccData		:= FALSE;
		tyLeaderToFollowerTag.bBypassMnlAccData	:= FALSE;
		tyLeaderToFollowerTag.bBlkDS			:= FALSE;
		tyLeaderToFollowerTag.bBlkUS			:= FALSE;
		tyLeaderToFollowerTag.bBypassWidthChk	:= TRUE;
		tyLeaderToFollowerTag.bSetTm			:= FALSE;
		tyLeaderToFollowerTag.dtTm				:= 0;
		tyLeaderToFollowerTag.uiTmZone			:= 0;
		tyLeaderToFollowerTag.usiRunTm			:= 0;
		tyLeaderToFollowerTag.bProdNameUSWarn	:= FALSE;
		tyLeaderToFollowerTag.bProdNameDSWarn	:= FALSE;
		tyLeaderToFollowerTag.bProdWidthUSWarn	:= FALSE;
		tyLeaderToFollowerTag.bProdWidthDSWarn	:= FALSE;
		tyLeaderToFollowerTag.bLeaderSeqCtrlInActive	:= FALSE;
	END_IF

	Act_Background_UpdtData;

	//FB
	fbFollower.tyLeaderToFollowerTag	:= tyLeaderToFollowerTag;
	fbFollower.sMcNm					:= g_tyMcParamCurr.sMcNm;
	fbFollower.sIPAddr					:= g_tyMcParamCurr.sIPAddr;
	fbFollower.bSectionLeader			:= g_tyMcParamCurr.bSectionLeader;
	fbFollower.sCurrProdRcpNm			:= p_tyCurrProdRcp.sRcpNm;
	fbFollower.diCurrProdWidthUS		:= p_tyCurrProdRcp.diWidthInUM;
	fbFollower.diCurrProdWidthDS		:= p_tyCurrProdRcp.diWidthInUM2;
	fbFollower.sCurrMagRcpNm			:= p_sCurrMagRcpNm;
	fbFollower.sUpdtLeaderProdRcpNm		:= p_tyFollower.tyUpdtProdRcp.sRcpNm;
	fbFollower.diUpdtLeaderProdWidthUS	:= p_tyFollower.tyUpdtProdRcp.diWidthInUM;
	fbFollower.diUpdtLeaderProdWidthDS	:= p_tyFollower.tyUpdtProdRcp.diWidthInUM2;
	fbFollower.sUpdtLeaderMagRcpNm		:= p_sMagRcpNm;
	fbFollower.bMnlAccDat				:= g_tyMcParamCurr.bMnlAccDat;
	fbFollower.bAWEn					:= (g_tyNtParamCurr.bAWPrep = TRUE) AND (g_tyMcParamCurr.bAWDis = FALSE);
	fbFollower.bUSWidthChkEn			:= g_tyNtParamCurr.bUSWidthChkPrep AND g_tyMcParamCurr.bUSWidthChkEn;
	fbFollower.bUSWidthChkSen			:= tylocalFollower.In.bUSWidthChkSen;
	fbFollower.bDSWidthChkEn			:= g_tyNtParamCurr.bDSWidthChkPrep AND g_tyMcParamCurr.bDSWidthChkEn;
	fbFollower.bDSWidthChkSen			:= tylocalFollower.In.bDSWidthChkSen;
	fbFollower.bProdWidthChk			:= g_tyNtParamCurr.bLFProdWidthChk;
	fbFollower.bProdRcpErr				:= bProdRcpErr;
	fbFollower.bMagRcpErr				:= bMagRcpErr;
	fbFollower.bSetTmErr				:= bSetTmErr;
	fbFollower.eCurrMachineStat			:= eCurrMachineStat;
	fbFollower.bProdChgOverActive		:= (g_tyAW.eStat = AWActGoWidthOff);
	fbFollower.bDBAOnWOAlign			:= g_tyMcParamCurr.bDBAOnWOAlign;

	fbFollower(bEn := TRUE);

	tyFollowerToLeaderTag	:= fbFollower.tyFollowerToLeaderTag;
	bProdAccDataReq			:= fbFollower.bProdAccDataReq OR (p_bInternalReqProdRcpDiff = TRUE) ;
	bMagAccDataReq			:= fbFollower.bMagAccDataReq;
	bAutoAccData			:= fbFollower.bAutoAccData;

	IF p_bInternalUse THEN
		bLeaderOnline			:= TRUE;
	ELSE
		bLeaderOnline			:= tylocalFollower.Out.tyLeaderInfo.bOnline;
	END_IF

	IF bLeaderOnline=FALSE THEN
		tylocalFollower.Out.bUSAllow				:= TRUE;
		tylocalFollower.Out.bDSAllow				:= TRUE;
		tylocalFollower.Out.bLdrSeqCtrlInActive	:= FALSE;
	ELSE
		tylocalFollower.Out.bUSAllow				:= fbFollower.bUSAllow AND (p_bInternalReqProdRcpDiff = FALSE);
		tylocalFollower.Out.bDSAllow				:= fbFollower.bDSAllow;
		tylocalFollower.Out.bLdrSeqCtrlInActive		:= tyLeaderToFollowerTag.bLeaderSeqCtrlInActive;
	END_IF

	fbOnlineChk.tyLeaderToFollowerTag	:= tyLeaderToFollowerTag;
	fbOnlineChk(bEn := TRUE);

	Act_Background_AccData;
	Act_Background_ChkRlsBrd;

	//Set Time
	IF EDGEPOS(tyLeaderToFollowerTag.bSetTm) THEN
		bSetTm	:= TRUE;
	END_IF

	IF bSetTm = TRUE THEN
		tylocalFollower.Out.eTimeAct	:= TimeActSetTime;

		IF (g_tyTime.eStat = TimeActSetTime) AND (g_tyTime.eMainStatus = Done) THEN
			tylocalFollower.Out.eTimeAct:= TimeActIdle;
			bSetTm			:= FALSE;
		ELSIF g_tyTime.eMainStatus = Error THEN
			tylocalFollower.Out.eTimeAct:= TimeActIdle;
			bSetTm			:= FALSE;
		END_IF
	END_IF

	bSetTmErr	:= g_tyTime.eMainStatus = Error;

	IF (tylocalFollower.Out.eStatus = Error) AND bRstErr THEN
		tylocalFollower.Out.eStatus		:= Idle;
		udiStatus	:= 0;
		bProdRcpErr	:= FALSE;
		bProdRcpErrNotExist	:= FALSE;
		bProdRcpErrWidthMismatch:= FALSE;
		bMagRcpErr	:= FALSE;
	END_IF

END_ACTION
```

#### Act_Background_AccData.st
```iecst
(** 2021-05-18 **)
ACTION Act_Background_AccData:
	//Product Accept Data Request
	CASE usiProdAccDatStep OF
		0:
			//Check Error & Request Accept Data
			// If Product Name/Width Error, Check In Background To Update Data
			IF ((eStatus <> Error) AND (bProdAccDataReq = TRUE)) OR bProdRcpErr THEN
				sReqProdRcpNm		:= tyLeaderToFollowerTag.sReqProdRcpNm;
				diReqProdRcpWidth	:= tyLeaderToFollowerTag.diReqProdRcpWidth;
				usiProdAccDatStep	:= 1;
			END_IF

			IF bLeaderOnline=FALSE THEN
				tyInfoData.sProgNm		:= '';
				tyInfoData.udiCode		:= 0;
				tyInfoData.eSeverity	:= AlmSeverityNA;
				tyInfoData.sAlmMsg		:= '';

				bProdRcpErr 			:= FALSE;
				bProdRcpErrNotExist		:= FALSE;
				bProdRcpErrWidthMismatch:= FALSE;
			END_IF

		1:
			IF p_bInternalUse THEN
				usiProdAccDatStep	:= 2;
			ELSE
				//Check In List Of Recipe
				FOR i := 1 TO 2000 DO
					IF sReqProdRcpNm = '' THEN
						EXIT;
					ELSIF sReqProdRcpNm = pa_tyProdRcpList[i].sRcpNm  THEN
						EXIT;
					END_IF
				END_FOR

				IF sReqProdRcpNm = pa_tyProdRcpList[i].sRcpNm AND diReqProdRcpWidth <> pa_tyProdRcpList[i].diWidthInUM THEN
					//Width Mismatch
					bProdRcpErr := TRUE;
					bProdRcpErrWidthMismatch:= TRUE;
					bProdRcpErrNotExist		:= FALSE;
					usiProdAccDatStep	:= 0;
				ELSIF i > 2000 THEN
					//Recipe Not Exist
					bProdRcpErr := TRUE;
					bProdRcpErrNotExist	:= TRUE;
					bProdRcpErrWidthMismatch:= FALSE;
					usiProdAccDatStep	:= 0;
				ELSE
					bProdRcpErr := FALSE;
					bProdRcpErrNotExist	:= FALSE;
					bProdRcpErrWidthMismatch:= FALSE;
					usiProdAccDatStep	:= 2;
				END_IF

				//Info Message
				IF bLeaderOnline=FALSE THEN
					tyInfoData.sProgNm		:= '';
					tyInfoData.udiCode		:= 0;
					tyInfoData.eSeverity	:= AlmSeverityNA;
					tyInfoData.sAlmMsg		:= '';

					bProdRcpErr 			:= FALSE;
					bProdRcpErrNotExist		:= FALSE;
					bProdRcpErrWidthMismatch:= FALSE;
				ELSE

					IF p_bInternalUse = FALSE THEN
						IF bLeaderInfo OR bFollowerInfo THEN
							tyInfoData.sProgNm		:= p_sProgNm;
							tyInfoData.udiCode		:= 10000;
							tyInfoData.eSeverity	:= AlmSeverityInfo;
							tyInfoData.sAlmMsg		:= p_sInfoMsg;
						ELSE
							tyInfoData.sProgNm		:= '';
							tyInfoData.udiCode		:= 0;
							tyInfoData.eSeverity	:= AlmSeverityNA;
							tyInfoData.sAlmMsg		:= '';
						END_IF
					ELSE
						IF p_sInfoMsg <> '' THEN
							tyInfoData.sProgNm		:= p_sProgNm;
							tyInfoData.udiCode		:= 10000;
							tyInfoData.eSeverity	:= AlmSeverityInfo;
							tyInfoData.sAlmMsg		:= p_sInfoMsg;
						ELSE
							tyInfoData.sProgNm		:= '';
							tyInfoData.udiCode		:= 0;
							tyInfoData.eSeverity	:= AlmSeverityNA;
							tyInfoData.sAlmMsg		:= '';
						END_IF

					END_IF
				END_IF
			END_IF
		2:
			//Manual Accept Data Check
			IF bProdAccDataReq = TRUE THEN
				IF bAutoAccData = FALSE THEN
					bProdAccDataMnl	:= TRUE;

					//Info Message
					IF bLeaderOnline=FALSE THEN
						tyInfoData.sProgNm		:= '';
						tyInfoData.udiCode		:= 0;
						tyInfoData.eSeverity	:= AlmSeverityNA;
						tyInfoData.sAlmMsg		:= '';
					ELSE
						IF p_sInfoMsg <> '' THEN
							tyInfoData.sProgNm		:= p_sProgNm;
							tyInfoData.udiCode		:= 10000;
							tyInfoData.eSeverity	:= AlmSeverityInfo;
							tyInfoData.sAlmMsg		:= p_sInfoMsg;
						ELSE
							tyInfoData.sProgNm		:= '';
							tyInfoData.udiCode		:= 0;
							tyInfoData.eSeverity	:= AlmSeverityNA;
							tyInfoData.sAlmMsg		:= '';
						END_IF
					END_IF

					IF p_bUIProdAccData = TRUE THEN
						p_bUIProdAccData := FALSE; //2023_07_26_Debug for Manual Accept Data automatically accept after product change many times
						bProdAccDataMnl		:= FALSE;
						usiProdAccDatStep	:= 3;
					END_IF
				ELSE
					bProdAccDataMnl		:= FALSE;
					p_bUIProdAccData := FALSE; //2023_07_26_Debug for Manual Accept Data automatically accept after product change many times
					usiProdAccDatStep	:= 3;
				END_IF
			ELSE
				bProdAccDataMnl		:= FALSE;
				usiProdAccDatStep	:= 6;
			END_IF

		3:
			//Accept New Recipe Condition
			IF bProdAccDataReq = TRUE THEN
				IF p_bAccNewRcpCond = TRUE THEN

					usiProdAccDatStep	:= 4;
				ELSE
					//Info Message
					IF bLeaderOnline=FALSE THEN
						tyInfoData.sProgNm		:= '';
						tyInfoData.udiCode		:= 0;
						tyInfoData.eSeverity	:= AlmSeverityNA;
						tyInfoData.sAlmMsg		:= '';
					ELSE
						IF p_sInfoMsg <> '' THEN
							tyInfoData.sProgNm		:= p_sProgNm;
							tyInfoData.udiCode		:= 10000;
							tyInfoData.eSeverity	:= AlmSeverityInfo;
							tyInfoData.sAlmMsg		:= p_sInfoMsg;
						ELSE
							tyInfoData.sProgNm		:= '';
							tyInfoData.udiCode		:= 0;
							tyInfoData.eSeverity	:= AlmSeverityNA;
							tyInfoData.sAlmMsg		:= '';
						END_IF
					END_IF
				END_IF
			ELSE
				usiProdAccDatStep	:= 6;
			END_IF

		4:
			//Accept New Recipe Name
			IF p_bInternalUse = TRUE THEN

				p_tyCurrProdRcp	:= p_tyInternalReqProdRcp;
				usiProdAccDatStep := 6;
			ELSE

				FOR i := 1 TO 2000 DO
					IF sReqProdRcpNm = '' THEN
						EXIT;
					ELSIF sReqProdRcpNm = pa_tyProdRcpList[i].sRcpNm THEN
						p_tyCurrProdRcp	:= pa_tyProdRcpList[i];

						EXIT;
					END_IF
				END_FOR

				IF i > 2000 THEN
					//Recipe Not Exist
					bProdRcpErr := TRUE;
					bProdRcpErrNotExist	:= TRUE;
				END_IF
				usiProdAccDatStep	:= 5;
			END_IF

		5:
			(* Add *)
			p_tyProdRcpCurrRcpWr 	:= p_tyCurrProdRcp;
			p_eLinkUIProdRcpAct 	:= ProdRcpActWriteCurrRcpParam;

			IF p_eProdRcpStat = ProdRcpActWriteCurrRcpParam AND p_eProdRcpStatus = Done THEN
				p_eLinkUIProdRcpAct := ProdRcpActIdle;
				usiProdAccDatStep := 6;
			END_IF

		6:
			//Clear Info Message
			tyInfoData.sProgNm		:= '';
			tyInfoData.udiCode		:= 0;
			tyInfoData.eSeverity	:= AlmSeverityNA;
			tyInfoData.sAlmMsg		:= '';

			usiProdAccDatStep	:= 0;

	END_CASE

END_ACTION
```

#### Act_Background_UpdtData.st
```iecst
ACTION Act_Background_UpdtData:

	//Update To Leader Recipe
	CASE usiProdUpdtDatStep OF
		0:
			//Update New Recipe Condition
			IF tylocalFollower.Out.tyUpdtProdRcp.sRcpNm <> '' THEN
				IF (p_tyCurrProdRcp.sRcpNm <> tylocalFollower.Out.tyUpdtProdRcp.sRcpNm) OR (p_bUpdtProdRcpDiff = TRUE) THEN
					IF p_bUpdtNewRcpCond = TRUE THEN
						usiProdUpdtDatStep	:= 1;
					END_IF
				END_IF
			ELSE
				tylocalFollower.Out.tyUpdtProdRcp	:= p_tyCurrProdRcp;
			END_IF

		1:
			//Manual Update Data Check
			IF p_bAutoUpdtData = FALSE THEN

				tylocalFollower.Out.bProdUpdtDataMnl		:= TRUE;

				IF p_bUIProdUpdtData = TRUE THEN
					tylocalFollower.Out.bProdUpdtDataMnl	:= FALSE;
					usiProdUpdtDatStep	:= 2;
				END_IF
			ELSE
				tylocalFollower.Out.bProdUpdtDataMnl	:= FALSE;
				usiProdUpdtDatStep	:= 2;
			END_IF

		2:
			//Update New Recipe
			tylocalFollower.Out.tyUpdtProdRcp	:= p_tyCurrProdRcp;

			usiProdUpdtDatStep	:= 0;

	END_CASE

END_ACTION
```

#### Act_InitGlobal.st
```iecst
(** 2019-06-27 **)
ACTION Act_InitGlobal:

	(* Always Change If Project Change *)

	//Pass Data To Link
	p_bLinkOpsRun ACCESS p_OpsRun;
	p_bLinkStartupRun ACCESS p_StartupRun;

	p_bLinkPshrConvHvBrd ACCESS p_PshrConvHvBrd;
	p_bLinkOpsTravLifULInitDone ACCESS p_OpsTravLifULInitDone;

	//Pass Data To Internal Use
	p_udiRstErr ACCESS p_RstErrReset;
	p_sIPAddr ACCESS p_HWInfoIPAddr;
	p_sMcNm ACCESS p_McParamMcNm;
	p_bUSWidthChkPrep ACCESS p_NtParamUSWidthChkPrep;
	p_bUSWidthChkEn ACCESS p_McParamUSWidthChkEn;
	p_bUSWidthChkSen ACCESS p_DIUSWidthChkSen;
	p_tyCurrProdRcp ACCESS p_ProdRcpCurrRcp1;
	p_tyInternalReqProdRcp ACCESS p_ProdRcpCurrRcp0;	//Follower 1 Assign With Default Recipe
	p_sProgNm ACCESS p_NtParamFollower1ProgNm;
	p_bNtSettingsLoadDone ACCESS p_StartupNtSettingsLoadDone;
	p_bWidth2Prep ACCESS p_NtParamLFWidth2Prep;

	p_bNtParamAutoRcpPrep ACCESS p_NtParamAutoRcpPrep;
	p_bMcParamAutoRcpDis  ACCESS p_McParamAutoRcpDisable;
	p_eNtParamAutoRcpPrecededBy ACCESS p_NtParamAutoRcpPrecededBy;
	(* Always Change If Project Change *)

END_ACTION
```

#### Act_InitLocal.st
```iecst
(** 2020-08-06 **)
ACTION Act_InitLocal:

	//Input Reference Link To Local Variable
	p_sMagRcpNm ACCESS ADR(sMagRcpNm);
	p_bUIProdAccData ACCESS ADR(bUIProdAccData);
	p_bUIProdUpdtData ACCESS ADR(bUIProdUpdtData);
	p_bUIMagAccData ACCESS ADR(bUIMagAccData);
	pa_tyProdRcpList ACCESS ADR(a_tyProdRcpList);
	p_tyCurrProdRcp ACCESS ADR(tyCurrProdRcp);
	p_sCurrMagRcpNm ACCESS ADR(sCurrMagRcpNm);
	p_bAccNewRcpCond ACCESS ADR(bAccNewRcpCond);
	p_bUpdtNewRcpCond ACCESS ADR(bUpdtNewRcpCond);
	p_bAutoUpdtData ACCESS ADR(bAutoUpdtData);
	p_sInfoMsg ACCESS ADR(sInfoMsg);
	p_bInternalUse ACCESS ADR(bInternalUse);
	p_tyInternalReqProdRcp ACCESS ADR(tyInternalReqProdRcp);
	p_bNewBrdEnteredCond ACCESS ADR(bNewBrdEnteredCond);
	p_bOldBrdExitedCond ACCESS ADR(bOldBrdExitedCond);
	p_bRlsBrd ACCESS ADR(bRlsBrd);
	p_bInternalReqProdRcpDiff ACCESS ADR(bInternalReqProdRcpDiff);
	p_bUpdtProdRcpDiff ACCESS ADR(bUpdtProdRcpDiff);
	p_bRlsBrdProdRcpDiff ACCESS ADR(bRlsBrdProdRcpDiff);
	p_tyFollower ACCESS ADR(tyFollower);

END_ACTION
```

#### Act_InputConfig.st
```iecst
(** 2019-06-27 **)
ACTION Act_InputConfig:

	p_tyCurrProdRcp ACCESS p_ProdRcpCurrRcp1;
	p_tyInternalReqProdRcp ACCESS p_ProdRcpCurrRcp0; //Follower 1 Assign With Default Recipe

	//US width check sensor selection
	tylocalFollower.In.bUSWidthChkSen := g_tyDInput.bUSWidthChkSen;

	//Link bPrep, bEn & bDis
	tylocalFollower.In.bDis	:= (g_tyStartUp.bRun = TRUE);
	IF g_tyNtParamCurr.bAutoRcpPrep AND NOT(g_tyMcParamCurr.bAutoRcpDisable) THEN
		CASE p_eNtParamAutoRcpPrecededBy OF
			PrecededBySelf:
				tylocalFollower.In.bPrep := FALSE;
			PrecededByF1:
				tylocalFollower.In.bPrep := TRUE;
		END_CASE
	ELSE
		tylocalFollower.In.bPrep := TRUE;
	END_IF

	//Temporary (Recipe No Save)
	IF p_tyCurrProdRcp.sRcpNm = '' AND p_tyCurrProdRcp.diWidthInUM = 0 THEN
		p_tyCurrProdRcp	:= p_tyInternalReqProdRcp;
	END_IF

	//Info Message
	p_sInfoMsg	:= '';

	//Accept New Recipe Condition (Before Loaded New Recipe)
	p_bAccNewRcpCond	:= (g_tyOps.bRun = TRUE) AND (g_tyOpsTravLifUL.bInitDone = TRUE) AND (g_tyPshrConv.bHvBrd = FALSE);

	//Update New Recipe Condition (After Loaded New Recipe)
	p_bUpdtNewRcpCond	:= TRUE;

	//Recipe Different
	p_bInternalReqProdRcpDiff	:= memcmp(ADR(p_tyCurrProdRcp) , ADR(p_tyInternalReqProdRcp) , SIZEOF(p_tyCurrProdRcp)) <> 0;
	p_bUpdtProdRcpDiff			:= memcmp(ADR(p_tyCurrProdRcp) , ADR(tylocalFollower.Out.tyUpdtProdRcp) , SIZEOF(p_tyCurrProdRcp)) <> 0;

END_ACTION
```

#### Act_Link.st
```iecst
(** 2019-07-04 **)
ACTION Act_Link:

	//Temporary (Recipe No Save)
	IF p_tyCurrProdRcp.sRcpNm = '' AND p_tyCurrProdRcp.diWidthInUM = 0 THEN
		p_tyCurrProdRcp	:= p_tyInternalReqProdRcp;
	END_IF

	//Info Message
	p_sInfoMsg	:= '';

	//Accept New Recipe Condition (Before Loaded New Recipe)
	p_bAccNewRcpCond	:= (p_bLinkOpsRun = TRUE) AND (p_bLinkOpsTravLifULInitDone = TRUE) AND (p_bLinkPshrConvHvBrd = FALSE);

	//Update New Recipe Condition (After Loaded New Recipe)
	p_bUpdtNewRcpCond	:= TRUE;

	//Recipe Different
	p_bInternalReqProdRcpDiff	:= memcmp(ADR(p_tyCurrProdRcp) , ADR(p_tyInternalReqProdRcp) , SIZEOF(p_tyCurrProdRcp)) <> 0;
	p_bUpdtProdRcpDiff			:= memcmp(ADR(p_tyCurrProdRcp) , ADR(tyUpdtProdRcp) , SIZEOF(p_tyCurrProdRcp)) <> 0;

END_ACTION
```

#### Act_LinkEn.st
```iecst
(** 2019-04-26 **)
ACTION Act_LinkEn:

	//Link bPrep, bEn & bDis
	p_bDis	:= (p_bLinkStartupRun = TRUE);
	IF p_bNtParamAutoRcpPrep AND NOT(p_bMcParamAutoRcpDis) THEN
		CASE p_eNtParamAutoRcpPrecededBy OF
			PrecededBySelf:
				p_bPrep := FALSE;
			PrecededByF1:
				p_bPrep := TRUE;
		END_CASE
	ELSE
		p_bPrep := TRUE;
	END_IF
END_ACTION
```

#### Act_Main_Disable.st
```iecst
(** 2020-09-21 **)
ACTION Act_Main_Disable:

	bUSAllow			:= TRUE;
	bDSAllow			:= TRUE;
	bProdAccDataMnl		:= FALSE;
	bProdUpdtDataMnl	:= FALSE;
	bMagAccDataMnl		:= FALSE;
	bWaitRlsBrd			:= FALSE;

	usiProdAccDatStep		:= 0;
	usiProdUpdtDatStep		:= 0;
	tyInfoData.sProgNm		:= '';
	tyInfoData.udiCode		:= 0;
	tyInfoData.eSeverity	:= AlmSeverityNA;
	tyInfoData.sAlmMsg		:= '';

	usiMagAccDatStep		:= 0;
	tyInfoData1.sProgNm		:= '';
	tyInfoData1.udiCode		:= 0;
	tyInfoData1.eSeverity	:= AlmSeverityNA;
	tyInfoData1.sAlmMsg		:= '';

	bSetTm		:= FALSE;

	eStatus		:= Idle;
	udiStatus	:= 0;
	bProdRcpErr	:= FALSE;
	bMagRcpErr	:= FALSE;
	bLeaderSeqCtrlInActive	:= FALSE;

	bProdRcpErrNotExist		:= FALSE;
	bProdRcpErrWidthMismatch:= FALSE;

END_ACTION
```

#### Init.st
```iecst
(** 2019-06-27 **)
PROGRAM _INIT
	//Physical Configuration
	bAutoUpdtData	:= TRUE;
	bInternalUse	:= TRUE;

	p_Follower1		:= ADR(tylocalFollower.Out);

END_PROGRAM
```

### Program Logical/LF/Follower2 (IEC, version 1.00.0) - 1.00.0 - NtHermes v5.00.0 , NtTCP v5.00.0 , NtMessage v5.00.0

#### Init.st - Change By Project
```iecst
(** 2019-06-27 **)
PROGRAM _INIT

		//Physical Configuration
	bAutoUpdtData	:= TRUE;
	bInternalUse	:= TRUE;

	p_Follower2		:= ADR(tylocalFollower.Out);

END_PROGRAM
```

#### Act_InitGlobal.st - Change By Project
```iecst
(** 2019-06-12 **)
ACTION Act_InitGlobal:

	(* Always Change If Project Change *)

	//Pass Data To Link
	p_bLinkStartupRun ACCESS p_StartupRun;

	p_bLinkOpsRun ACCESS p_OpsRun;
	p_eLinkNtParamProjMag ACCESS p_NtParamProjMag;
	p_bLinkNtParamProjMagConv1Prep ACCESS p_NtParamProjMag1ConvPrep;
	p_bLinkNtParamProjMagConv2Prep ACCESS p_NtParamProjMag2ConvPrep;
	p_bLinkNtParamProjMagConv3Prep ACCESS p_NtParamProjMag3ConvPrep;
	p_bLinkBffr1MagRemoved ACCESS p_Buffer1MagRemoved;
	p_bLinkBffr2MagRemoved ACCESS p_Buffer2MagRemoved;
	p_bLinkBffr3MagRemoved ACCESS p_Buffer3MagRemoved;
//	p_bLinkOpsMagUL1InitDone ACCESS p_OpsMagUL1InitDone;
//	p_bLinkOpsMagUL2InitDone ACCESS p_OpsMagUL2InitDone;
//	p_bLinkOpsMagUL3InitDone ACCESS p_OpsMagUL3InitDone;
	p_bLinkOpsMagConvUL1InitDone ACCESS p_OpsMagConvUL1InitDone;
	p_bLinkOpsMagConvUL2InitDone ACCESS p_OpsMagConvUL2InitDone;
	p_bLinkOpsMagConvUL3InitDone ACCESS p_OpsMagConvUL3InitDone;

	//Pass Data To Internal Use
	p_udiRstErr ACCESS p_RstErrReset;
	p_tyCurrProdRcp ACCESS p_ProdRcpCurrRcp2;
	p_tyInternalReqProdRcp ACCESS p_Follower1UpdtProdRcp;	//Follower 2 Assign With Follower 1 Recipe
	p_sProgNm ACCESS p_NtParamFollower2ProgNm;
	p_bNtSettingsLoadDone ACCESS p_StartupNtSettingsLoadDone;
	p_bWidth2Prep ACCESS p_NtParamLFWidth2Prep;

	p_bNtParamAutoRcpPrep ACCESS p_NtParamAutoRcpPrep;
	p_bMcParamAutoRcpDis  ACCESS p_McParamAutoRcpDisable;
	p_bNtParamAutoRcpF1ArbitraryType ACCESS p_NtParamAutoRcpF1ArbitraryType;
//	p_bPrep ACCESS ;
	(* Always Change If Project Change *)

END_ACTION
```

#### InputRef_Link.var - Change By Project
```iecst
(*2019-05-07*)
(**)
VAR
	p_bLinkStartupRun : REFERENCE TO BOOL;
END_VAR
(**)
VAR
	p_bLinkOpsRun : REFERENCE TO BOOL;
	p_eLinkNtParamProjMag : REFERENCE TO eULMag;
	p_bLinkNtParamProjMagConv1Prep : REFERENCE TO BOOL;
	p_bLinkNtParamProjMagConv2Prep : REFERENCE TO BOOL;
	p_bLinkNtParamProjMagConv3Prep : REFERENCE TO BOOL;
	p_bLinkBffr1MagRemoved : REFERENCE TO BOOL;
	p_bLinkBffr2MagRemoved : REFERENCE TO BOOL;
	p_bLinkBffr3MagRemoved : REFERENCE TO BOOL;
	p_bLinkOpsMagUL1InitDone : REFERENCE TO BOOL;
	p_bLinkOpsMagUL2InitDone : REFERENCE TO BOOL;
	p_bLinkOpsMagUL3InitDone : REFERENCE TO BOOL;
	p_bLinkOpsMagConvUL1InitDone : REFERENCE TO BOOL;
	p_bLinkOpsMagConvUL2InitDone : REFERENCE TO BOOL;
	p_bLinkOpsMagConvUL3InitDone : REFERENCE TO BOOL;
END_VAR
(**)
VAR
	bOpsInitDone : BOOL;
	p_eLinkUIProdRcpAct : REFERENCE TO eProdRcpAction;
	p_eProdRcpStat : REFERENCE TO eProdRcpAction;
	p_eProdRcpStatus : REFERENCE TO eFBStatus;
	p_tyProdRcpCurrRcpWr : REFERENCE TO tyProdRcpParam;
END_VAR
```

#### Act_LinkEn.st - Change By Project
```iecst
(** 2019-04-26 **)
ACTION Act_LinkEn:

	//Link bPrep, bEn & bDis
	p_bDis	:= (p_bLinkStartupRun = TRUE);

	p_bPrep := NOT(p_bNtParamAutoRcpPrep AND NOT(p_bNtParamAutoRcpF1ArbitraryType)) OR p_bMcParamAutoRcpDis;
END_ACTION
```
